LIN {X 0,Y 608.989,Z 328.359,A -85,B 0,C 180,E1 28957.914,E2 28957.914} C_VEL
LIN {X 0,Y 609.026,Z 328.336,A -85,B 0,C 180,E1 28955.043,E2 28955.043} C_VEL
LIN {X 0,Y 608.99,Z 328.372,A -85,B 0,C 180,E1 28951.886,E2 28951.886} C_VEL
LIN {X 0,Y 608.992,Z 328.336,A -85,B 0,C 180,E1 28949.168,E2 28949.168} C_VEL
LIN {X 0,Y 608.991,Z 328.34,A -85,B 0,C 180,E1 28945.952,E2 28945.952} C_VEL
LIN {X 0,Y 609.049,Z 328.447,A -85,B 0,C 180,E1 28944.672,E2 28944.672} C_VEL
LIN {X 0,Y 610.191,Z 331.571,A -85,B 0,C 180,E1 28944.457,E2 28944.457} C_VEL
LIN {X 0,Y 612.692,Z 334.142,A -85,B 0,C 180,E1 28944.077,E2 28944.077} C_VEL
LIN {X 0,Y 613.552,Z 335.036,A -85,B 0,C 180,E1 28943.948,E2 28943.948} C_VEL
LIN {X 0,Y 616.041,Z 338.824,A -85,B 0,C 180,E1 28943.555,E2 28943.555} C_VEL
LIN {X 0,Y 618.268,Z 341.03,A -85,B 0,C 180,E1 28943.231,E2 28943.231} C_VEL
LIN {X 0,Y 621.516,Z 345.277,A -85,B 0,C 180,E1 28942.749,E2 28942.749} C_VEL
LIN {X 0,Y 626.243,Z 351.226,A -85,B 0,C 180,E1 28942.069,E2 28942.069} C_VEL
LIN {X 0,Y 641.999,Z 372.195,A -85,B 0,C 180,E1 28939.923,E2 28939.923} C_VEL
LIN {X 0,Y 650.667,Z 384.496,A -85,B 0,C 180,E1 28938.812,E2 28938.812} C_VEL
LIN {X 0,Y 648.081,Z 493.94,A -85,B 0,C 180,E1 28937.285,E2 28937.285} C_VEL
LIN {X 0,Y 647.227,Z 501.644,A -85,B 0,C 180,E1 28937.244,E2 28937.244} C_VEL
LIN {X 0,Y 642.505,Z 522.314,A -85,B 0,C 180,E1 28937.368,E2 28937.368} C_VEL
LIN {X 0,Y 641.836,Z 528.923,A -85,B 0,C 180,E1 28937.326,E2 28937.326} C_VEL
LIN {X 0,Y 636.639,Z 753.083,A -85,B 0,C 180,E1 28934.254,E2 28934.254} C_VEL
LIN {X 0,Y 635.306,Z 802.32,A -85,B 0,C 180,E1 28933.564,E2 28933.564} C_VEL
LIN {X 0,Y 633.786,Z 830.264,A -85,B 0,C 180,E1 28933.009,E2 28933.009} C_VEL
LIN {X 0,Y 632.226,Z 852.784,A -85,B 0,C 180,E1 28932.423,E2 28932.423} C_VEL
LIN {X 0,Y 630.535,Z 873.77,A -85,B 0,C 180,E1 28931.759,E2 28931.759} C_VEL
LIN {X 0,Y 628.677,Z 894.198,A -85,B 0,C 180,E1 28930.999,E2 28930.999} C_VEL
LIN {X 0,Y 626.241,Z 918.774,A -85,B 0,C 180,E1 28929.929,E2 28929.929} C_VEL
LIN {X 0,Y 623.465,Z 943.532,A -85,B 0,C 180,E1 28928.644,E2 28928.644} C_VEL
LIN {X 0,Y 621.108,Z 963.324,A -85,B 0,C 180,E1 28927.471,E2 28927.471} C_VEL
LIN {X 0,Y 618.751,Z 982.414,A -85,B 0,C 180,E1 28926.201,E2 28926.201} C_VEL
LIN {X 0,Y 616.012,Z 1004.354,A -85,B 0,C 180,E1 28924.561,E2 28924.561} C_VEL
LIN {X 0,Y 613.186,Z 1025.937,A -85,B 0,C 180,E1 28922.71,E2 28922.71} C_VEL
LIN {X 0,Y 611.026,Z 1042.889,A -85,B 0,C 180,E1 28921.082,E2 28921.082} C_VEL
LIN {X 0,Y 608.96,Z 1059.696,A -85,B 0,C 180,E1 28919.294,E2 28919.294} C_VEL
LIN {X 0,Y 606.611,Z 1079.55,A -85,B 0,C 180,E1 28916.906,E2 28916.906} C_VEL
LIN {X 0,Y 604.981,Z 1094.558,A -85,B 0,C 180,E1 28914.855,E2 28914.855} C_VEL
LIN {X 0,Y 603.522,Z 1109.273,A -85,B 0,C 180,E1 28912.604,E2 28912.604} C_VEL
LIN {X 0,Y 602.265,Z 1123.493,A -85,B 0,C 180,E1 28910.1,E2 28910.1} C_VEL
LIN {X 0,Y 601.47,Z 1133.871,A -85,B 0,C 180,E1 28908.011,E2 28908.011} C_VEL
LIN {X 0,Y 600.869,Z 1143.337,A -85,B 0,C 180,E1 28905.837,E2 28905.837} C_VEL
LIN {X 0,Y 600.412,Z 1152.859,A -85,B 0,C 180,E1 28903.286,E2 28903.286} C_VEL
LIN {X 0,Y 600.121,Z 1160.474,A -85,B 0,C 180,E1 28900.755,E2 28900.755} C_VEL
LIN {X 0,Y 600.004,Z 1166.042,A -85,B 0,C 180,E1 28898.433,E2 28898.433} C_VEL
LIN {X 0,Y 599.936,Z 1170.564,A -85,B 0,C 180,E1 28895.931,E2 28895.931} C_VEL
LIN {X 0,Y 599.914,Z 1173.552,A -85,B 0,C 180,E1 28893.344,E2 28893.344} C_VEL
LIN {X 0,Y 599.91,Z 1174.749,A -85,B 0,C 180,E1 28891.05,E2 28891.05} C_VEL
LIN {X 0,Y 599.907,Z 1174.793,A -85,B 0,C 180,E1 28889.045,E2 28889.045} C_VEL
LIN {X 0,Y 599.913,Z 1173.823,A -85,B 0,C 180,E1 28886.943,E2 28886.943} C_VEL
LIN {X 0,Y 599.923,Z 1171.362,A -85,B 0,C 180,E1 28884.549,E2 28884.549} C_VEL
LIN {X 0,Y 599.991,Z 1166.847,A -85,B 0,C 180,E1 28881.855,E2 28881.855} C_VEL
LIN {X 0,Y 600.108,Z 1161.212,A -85,B 0,C 180,E1 28879.437,E2 28879.437} C_VEL
LIN {X 0,Y 600.366,Z 1154.109,A -85,B 0,C 180,E1 28877.007,E2 28877.007} C_VEL
LIN {X 0,Y 600.82,Z 1144.11,A -85,B 0,C 180,E1 28874.261,E2 28874.261} C_VEL
LIN {X 0,Y 601.415,Z 1134.739,A -85,B 0,C 180,E1 28872.088,E2 28872.088} C_VEL
LIN {X 0,Y 602.187,Z 1124.472,A -85,B 0,C 180,E1 28869.999,E2 28869.999} C_VEL
LIN {X 0,Y 603.358,Z 1111.046,A -85,B 0,C 180,E1 28867.595,E2 28867.595} C_VEL
LIN {X 0,Y 604.905,Z 1095.289,A -85,B 0,C 180,E1 28865.16,E2 28865.16} C_VEL
LIN {X 0,Y 606.386,Z 1081.406,A -85,B 0,C 180,E1 28863.247,E2 28863.247} C_VEL
LIN {X 0,Y 608.474,Z 1064.093,A -85,B 0,C 180,E1 28861.112,E2 28861.112} C_VEL
LIN {X 0,Y 610.807,Z 1044.692,A -85,B 0,C 180,E1 28859.01,E2 28859.01} C_VEL
LIN {X 0,Y 612.933,Z 1027.84,A -85,B 0,C 180,E1 28857.375,E2 28857.375} C_VEL
LIN {X 0,Y 615.269,Z 1009.673,A -85,B 0,C 180,E1 28855.787,E2 28855.787} C_VEL
LIN {X 0,Y 618.361,Z 985.78,A -85,B 0,C 180,E1 28853.945,E2 28853.945} C_VEL
LIN {X 0,Y 620.892,Z 965.162,A -85,B 0,C 180,E1 28852.555,E2 28852.555} C_VEL
LIN {X 0,Y 623.12,Z 946.531,A -85,B 0,C 180,E1 28851.436,E2 28851.436} C_VEL
LIN {X 0,Y 625.266,Z 927.631,A -85,B 0,C 180,E1 28850.425,E2 28850.425} C_VEL
LIN {X 0,Y 627.464,Z 906.92,A -85,B 0,C 180,E1 28849.448,E2 28849.448} C_VEL
LIN {X 0,Y 629.999,Z 880.352,A -85,B 0,C 180,E1 28848.378,E2 28848.378} C_VEL
LIN {X 0,Y 631.987,Z 855.974,A -85,B 0,C 180,E1 28847.58,E2 28847.58} C_VEL
LIN {X 0,Y 633.509,Z 834.338,A -85,B 0,C 180,E1 28846.999,E2 28846.999} C_VEL
LIN {X 0,Y 634.765,Z 812.654,A -85,B 0,C 180,E1 28846.532,E2 28846.532} C_VEL
LIN {X 0,Y 635.903,Z 785.947,A -85,B 0,C 180,E1 28846.1,E2 28846.1} C_VEL
LIN {X 0,Y 641.062,Z 561.333,A -85,B 0,C 180,E1 28843.033,E2 28843.033} C_VEL
LIN {X 0,Y 645.263,Z 388.229,A -85,B 0,C 180,E1 28840.604,E2 28840.604} C_VEL
LIN {X 0,Y 633.126,Z 371.566,A -85,B 0,C 180,E1 28839.002,E2 28839.002} C_VEL
LIN {X 0,Y 622.468,Z 357.45,A -85,B 0,C 180,E1 28837.503,E2 28837.503} C_VEL
LIN {X 0,Y 617.121,Z 350.737,A -85,B 0,C 180,E1 28836.718,E2 28836.718} C_VEL
LIN {X 0,Y 613.975,Z 346.647,A -85,B 0,C 180,E1 28836.24,E2 28836.24} C_VEL
LIN {X 0,Y 610.658,Z 342.52,A -85,B 0,C 180,E1 28835.728,E2 28835.728} C_VEL
LIN {X 0,Y 609.495,Z 340.975,A -85,B 0,C 180,E1 28835.544,E2 28835.544} C_VEL
LIN {X 0,Y 606.547,Z 337.524,A -85,B 0,C 180,E1 28835.079,E2 28835.079} C_VEL
LIN {X 0,Y 605.262,Z 335.42,A -85,B 0,C 180,E1 28834.861,E2 28834.861} C_VEL
LIN {X 0,Y 602.43,Z 332.951,A -85,B 0,C 180,E1 28834.419,E2 28834.419} C_VEL
LIN {X 0,Y 601.129,Z 329.909,A -85,B 0,C 180,E1 28834.172,E2 28834.172} C_VEL
LIN {X 0,Y 601.037,Z 329.326,A -85,B 0,C 180,E1 28834.133,E2 28834.133} C_VEL
LIN {X 0,Y 601.047,Z 329.325,A -85,B 0,C 180,E1 28830.823,E2 28830.823} C_VEL
LIN {X 0,Y 601.042,Z 329.362,A -85,B 0,C 180,E1 28828.086,E2 28828.086} C_VEL
LIN {X 0,Y 601.077,Z 329.323,A -85,B 0,C 180,E1 28824.889,E2 28824.889} C_VEL
LIN {X 0,Y 601.044,Z 329.352,A -85,B 0,C 180,E1 28822.084,E2 28822.084} C_VEL
LIN {X 0,Y 601.118,Z 329.326,A -85,B 0,C 180,E1 28819.028,E2 28819.028} C_VEL
LIN {X 0,Y 601.048,Z 329.337,A -85,B 0,C 180,E1 28816.031,E2 28816.031} C_VEL
LIN {X 0,Y 601.129,Z 329.335,A -85,B 0,C 180,E1 28812.977,E2 28812.977} C_VEL
LIN {X 0,Y 601.054,Z 329.33,A -85,B 0,C 180,E1 28809.963,E2 28809.963} C_VEL
LIN {X 0,Y 601.14,Z 329.337,A -85,B 0,C 180,E1 28806.878,E2 28806.878} C_VEL
LIN {X 0,Y 601.059,Z 329.328,A -85,B 0,C 180,E1 28803.815,E2 28803.815} C_VEL
LIN {X 0,Y 601.136,Z 329.337,A -85,B 0,C 180,E1 28800.762,E2 28800.762} C_VEL
LIN {X 0,Y 601.067,Z 329.327,A -85,B 0,C 180,E1 28797.712,E2 28797.712} C_VEL
LIN {X 0,Y 601.134,Z 329.338,A -85,B 0,C 180,E1 28794.655,E2 28794.655} C_VEL
LIN {X 0,Y 601.073,Z 329.323,A -85,B 0,C 180,E1 28791.582,E2 28791.582} C_VEL
LIN {X 0,Y 601.137,Z 329.345,A -85,B 0,C 180,E1 28788.486,E2 28788.486} C_VEL
LIN {X 0,Y 601.077,Z 329.316,A -85,B 0,C 180,E1 28785.354,E2 28785.354} C_VEL
LIN {X 0,Y 601.14,Z 329.351,A -85,B 0,C 180,E1 28782.279,E2 28782.279} C_VEL
LIN {X 0,Y 601.085,Z 329.318,A -85,B 0,C 180,E1 28779.146,E2 28779.146} C_VEL
LIN {X 0,Y 601.136,Z 329.331,A -85,B 0,C 180,E1 28776.055,E2 28776.055} C_VEL
LIN {X 0,Y 601.096,Z 329.352,A -85,B 0,C 180,E1 28772.884,E2 28772.884} C_VEL
LIN {X 0,Y 601.136,Z 329.316,A -85,B 0,C 180,E1 28769.682,E2 28769.682} C_VEL
LIN {X 0,Y 601.155,Z 329.494,A -85,B 0,C 180,E1 28767.73,E2 28767.73} C_VEL
LIN {X 0,Y 602.27,Z 332.603,A -85,B 0,C 180,E1 28767.233,E2 28767.233} C_VEL
LIN {X 0,Y 603.588,Z 334.345,A -85,B 0,C 180,E1 28766.861,E2 28766.861} C_VEL
LIN {X 0,Y 605.493,Z 338.277,A -85,B 0,C 180,E1 28766.185,E2 28766.185} C_VEL
LIN {X 0,Y 610.426,Z 347.698,A -85,B 0,C 180,E1 28764.617,E2 28764.617} C_VEL
LIN {X 0,Y 625.354,Z 368.362,A -85,B 0,C 180,E1 28762.368,E2 28762.368} C_VEL
LIN {X 0,Y 641.991,Z 392.611,A -85,B 0,C 180,E1 28760.082,E2 28760.082} C_VEL
LIN {X 0,Y 645.613,Z 398.452,A -85,B 0,C 180,E1 28759.605,E2 28759.605} C_VEL
LIN {X 0,Y 640.632,Z 604.673,A -85,B 0,C 180,E1 28756.729,E2 28756.729} C_VEL
LIN {X 0,Y 635.662,Z 822.347,A -85,B 0,C 180,E1 28753.759,E2 28753.759} C_VEL
LIN {X 0,Y 634.658,Z 844.67,A -85,B 0,C 180,E1 28753.384,E2 28753.384} C_VEL
LIN {X 0,Y 633.39,Z 866.16,A -85,B 0,C 180,E1 28752.912,E2 28752.912} C_VEL
LIN {X 0,Y 631.712,Z 889.713,A -85,B 0,C 180,E1 28752.266,E2 28752.266} C_VEL
LIN {X 0,Y 629.333,Z 917.45,A -85,B 0,C 180,E1 28751.31,E2 28751.31} C_VEL
LIN {X 0,Y 627.184,Z 939.464,A -85,B 0,C 180,E1 28750.394,E2 28750.394} C_VEL
LIN {X 0,Y 625.147,Z 958.693,A -85,B 0,C 180,E1 28749.476,E2 28749.476} C_VEL
LIN {X 0,Y 622.955,Z 977.953,A -85,B 0,C 180,E1 28748.438,E2 28748.438} C_VEL
LIN {X 0,Y 620.583,Z 997.794,A -85,B 0,C 180,E1 28747.234,E2 28747.234} C_VEL
LIN {X 0,Y 617.516,Z 1022.228,A -85,B 0,C 180,E1 28745.54,E2 28745.54} C_VEL
LIN {X 0,Y 614.967,Z 1041.908,A -85,B 0,C 180,E1 28743.981,E2 28743.981} C_VEL
LIN {X 0,Y 612.783,Z 1059.055,A -85,B 0,C 180,E1 28742.467,E2 28742.467} C_VEL
LIN {X 0,Y 610.531,Z 1077.071,A -85,B 0,C 180,E1 28740.704,E2 28740.704} C_VEL
LIN {X 0,Y 608.06,Z 1097.15,A -85,B 0,C 180,E1 28738.48,E2 28738.48} C_VEL
LIN {X 0,Y 606.258,Z 1112.619,A -85,B 0,C 180,E1 28736.547,E2 28736.547} C_VEL
LIN {X 0,Y 604.639,Z 1127.891,A -85,B 0,C 180,E1 28734.419,E2 28734.419} C_VEL
LIN {X 0,Y 603.102,Z 1143.702,A -85,B 0,C 180,E1 28731.902,E2 28731.902} C_VEL
LIN {X 0,Y 602.121,Z 1155.273,A -85,B 0,C 180,E1 28729.801,E2 28729.801} C_VEL
LIN {X 0,Y 601.343,Z 1165.909,A -85,B 0,C 180,E1 28727.615,E2 28727.615} C_VEL
LIN {X 0,Y 600.69,Z 1177.02,A -85,B 0,C 180,E1 28724.951,E2 28724.951} C_VEL
LIN {X 0,Y 600.299,Z 1185.324,A -85,B 0,C 180,E1 28722.557,E2 28722.557} C_VEL
LIN {X 0,Y 600.092,Z 1191.863,A -85,B 0,C 180,E1 28720.27,E2 28720.27} C_VEL
LIN {X 0,Y 599.973,Z 1197.542,A -85,B 0,C 180,E1 28717.758,E2 28717.758} C_VEL
LIN {X 0,Y 599.926,Z 1201.663,A -85,B 0,C 180,E1 28715.163,E2 28715.163} C_VEL
LIN {X 0,Y 599.915,Z 1203.927,A -85,B 0,C 180,E1 28712.866,E2 28712.866} C_VEL
LIN {X 0,Y 599.895,Z 1204.849,A -85,B 0,C 180,E1 28710.668,E2 28710.668} C_VEL
LIN {X 0,Y 599.908,Z 1204.623,A -85,B 0,C 180,E1 28708.376,E2 28708.376} C_VEL
LIN {X 0,Y 599.918,Z 1202.789,A -85,B 0,C 180,E1 28705.795,E2 28705.795} C_VEL
LIN {X 0,Y 599.944,Z 1199.513,A -85,B 0,C 180,E1 28703.375,E2 28703.375} C_VEL
LIN {X 0,Y 600.014,Z 1195.106,A -85,B 0,C 180,E1 28701.085,E2 28701.085} C_VEL
LIN {X 0,Y 600.197,Z 1188.477,A -85,B 0,C 180,E1 28698.469,E2 28698.469} C_VEL
LIN {X 0,Y 600.504,Z 1180.572,A -85,B 0,C 180,E1 28696.029,E2 28696.029} C_VEL
LIN {X 0,Y 600.938,Z 1172.306,A -85,B 0,C 180,E1 28693.868,E2 28693.868} C_VEL
LIN {X 0,Y 601.566,Z 1162.692,A -85,B 0,C 180,E1 28691.691,E2 28691.691} C_VEL
LIN {X 0,Y 602.621,Z 1149.398,A -85,B 0,C 180,E1 28689.092,E2 28689.092} C_VEL
LIN {X 0,Y 603.843,Z 1135.741,A -85,B 0,C 180,E1 28686.791,E2 28686.791} C_VEL
LIN {X 0,Y 605.279,Z 1121.578,A -85,B 0,C 180,E1 28684.669,E2 28684.669} C_VEL
LIN {X 0,Y 607.376,Z 1103.066,A -85,B 0,C 180,E1 28682.233,E2 28682.233} C_VEL
LIN {X 0,Y 609.273,Z 1086.965,A -85,B 0,C 180,E1 28680.359,E2 28680.359} C_VEL
LIN {X 0,Y 611.356,Z 1070.397,A -85,B 0,C 180,E1 28678.622,E2 28678.622} C_VEL
LIN {X 0,Y 614.09,Z 1049.297,A -85,B 0,C 180,E1 28676.647,E2 28676.647} C_VEL
LIN {X 0,Y 616.657,Z 1028.87,A -85,B 0,C 180,E1 28674.969,E2 28674.969} C_VEL
LIN {X 0,Y 619.038,Z 1009.978,A -85,B 0,C 180,E1 28673.583,E2 28673.583} C_VEL
LIN {X 0,Y 621.631,Z 988.944,A -85,B 0,C 180,E1 28672.207,E2 28672.207} C_VEL
LIN {X 0,Y 624.587,Z 963.722,A -85,B 0,C 180,E1 28670.778,E2 28670.778} C_VEL
LIN {X 0,Y 626.818,Z 942.858,A -85,B 0,C 180,E1 28669.757,E2 28669.757} C_VEL
LIN {X 0,Y 628.829,Z 922.588,A -85,B 0,C 180,E1 28668.892,E2 28668.892} C_VEL
LIN {X 0,Y 630.688,Z 901.904,A -85,B 0,C 180,E1 28668.131,E2 28668.131} C_VEL
LIN {X 0,Y 632.495,Z 879.261,A -85,B 0,C 180,E1 28667.429,E2 28667.429} C_VEL
LIN {X 0,Y 634.363,Z 850.617,A -85,B 0,C 180,E1 28666.733,E2 28666.733} C_VEL
LIN {X 0,Y 635.496,Z 826.763,A -85,B 0,C 180,E1 28666.307,E2 28666.307} C_VEL
LIN {X 0,Y 639.752,Z 643.039,A -85,B 0,C 180,E1 28663.798,E2 28663.798} C_VEL
LIN {X 0,Y 644.902,Z 427.367,A -85,B 0,C 180,E1 28660.804,E2 28660.804} C_VEL
LIN {X 0,Y 645.53,Z 398.043,A -85,B 0,C 180,E1 28660.38,E2 28660.38} C_VEL
LIN {X 0,Y 628.947,Z 373.409,A -85,B 0,C 180,E1 28658.144,E2 28658.144} C_VEL
LIN {X 0,Y 616.881,Z 356.682,A -85,B 0,C 180,E1 28656.388,E2 28656.388} C_VEL
LIN {X 0,Y 609.775,Z 346.816,A -85,B 0,C 180,E1 28655.254,E2 28655.254} C_VEL
LIN {X 0,Y 605.475,Z 338.255,A -85,B 0,C 180,E1 28653.816,E2 28653.816} C_VEL
LIN {X 0,Y 603.577,Z 334.304,A -85,B 0,C 180,E1 28653.14,E2 28653.14} C_VEL
LIN {X 0,Y 601.478,Z 330.889,A -85,B 0,C 180,E1 28652.477,E2 28652.477} C_VEL
LIN {X 0,Y 601.135,Z 329.344,A -85,B 0,C 180,E1 28652.215,E2 28652.215} C_VEL
LIN {X 0,Y 601.094,Z 329.323,A -85,B 0,C 180,E1 28649.06,E2 28649.06} C_VEL
LIN {X 0,Y 601.134,Z 329.317,A -85,B 0,C 180,E1 28645.942,E2 28645.942} C_VEL
LIN {X 0,Y 601.093,Z 329.356,A -85,B 0,C 180,E1 28642.804,E2 28642.804} C_VEL
LIN {X 0,Y 601.133,Z 329.312,A -85,B 0,C 180,E1 28639.633,E2 28639.633} C_VEL
LIN {X 0,Y 601.089,Z 329.346,A -85,B 0,C 180,E1 28636.526,E2 28636.526} C_VEL
LIN {X 0,Y 601.127,Z 329.33,A -85,B 0,C 180,E1 28633.337,E2 28633.337} C_VEL
LIN {X 0,Y 601.082,Z 329.332,A -85,B 0,C 180,E1 28630.35,E2 28630.35} C_VEL
LIN {X 0,Y 601.122,Z 329.339,A -85,B 0,C 180,E1 28627.167,E2 28627.167} C_VEL
LIN {X 0,Y 601.077,Z 329.327,A -85,B 0,C 180,E1 28624.197,E2 28624.197} C_VEL
LIN {X 0,Y 601.109,Z 329.345,A -85,B 0,C 180,E1 28620.953,E2 28620.953} C_VEL
LIN {X 0,Y 601.07,Z 329.328,A -85,B 0,C 180,E1 28618.093,E2 28618.093} C_VEL
LIN {X 0,Y 601.117,Z 329.342,A -85,B 0,C 180,E1 28614.942,E2 28614.942} C_VEL
LIN {X 0,Y 601.061,Z 329.33,A -85,B 0,C 180,E1 28612.064,E2 28612.064} C_VEL
LIN {X 0,Y 601.124,Z 329.341,A -85,B 0,C 180,E1 28608.918,E2 28608.918} C_VEL
LIN {X 0,Y 601.056,Z 329.325,A -85,B 0,C 180,E1 28605.888,E2 28605.888} C_VEL
LIN {X 0,Y 601.122,Z 329.349,A -85,B 0,C 180,E1 28602.778,E2 28602.778} C_VEL
LIN {X 0,Y 601.049,Z 329.318,A -85,B 0,C 180,E1 28599.755,E2 28599.755} C_VEL
LIN {X 0,Y 601.122,Z 329.353,A -85,B 0,C 180,E1 28596.657,E2 28596.657} C_VEL
LIN {X 0,Y 601.044,Z 329.328,A -85,B 0,C 180,E1 28593.629,E2 28593.629} C_VEL
LIN {X 0,Y 601.127,Z 329.322,A -85,B 0,C 180,E1 28590.614,E2 28590.614} C_VEL
LIN {X 0,Y 601.039,Z 329.365,A -85,B 0,C 180,E1 28587.61,E2 28587.61} C_VEL
LIN {X 0,Y 601.062,Z 329.488,A -85,B 0,C 180,E1 28585.75,E2 28585.75} C_VEL
LIN {X 0,Y 602.122,Z 332.471,A -85,B 0,C 180,E1 28585.538,E2 28585.538} C_VEL
LIN {X 0,Y 604.551,Z 334.996,A -85,B 0,C 180,E1 28585.149,E2 28585.149} C_VEL
LIN {X 0,Y 605.796,Z 336.054,A -85,B 0,C 180,E1 28584.957,E2 28584.957} C_VEL
LIN {X 0,Y 608.346,Z 339.929,A -85,B 0,C 180,E1 28584.535,E2 28584.535} C_VEL
LIN {X 0,Y 610.44,Z 342.145,A -85,B 0,C 180,E1 28584.214,E2 28584.214} C_VEL
LIN {X 0,Y 613.674,Z 346.372,A -85,B 0,C 180,E1 28583.711,E2 28583.711} C_VEL
LIN {X 0,Y 615.392,Z 348.396,A -85,B 0,C 180,E1 28583.452,E2 28583.452} C_VEL
LIN {X 0,Y 620.152,Z 354.623,A -85,B 0,C 180,E1 28582.74,E2 28582.74} C_VEL
LIN {X 0,Y 627.738,Z 364.357,A -85,B 0,C 180,E1 28581.653,E2 28581.653} C_VEL
LIN {X 0,Y 638.992,Z 379.544,A -85,B 0,C 180,E1 28580.12,E2 28580.12} C_VEL
LIN {X 0,Y 645.334,Z 388.642,A -85,B 0,C 180,E1 28579.292,E2 28579.292} C_VEL
LIN {X 0,Y 641.836,Z 528.923,A -85,B 0,C 180,E1 28577.326,E2 28577.326} C_VEL
LIN {X 0,Y 640.974,Z 536.628,A -85,B 0,C 180,E1 28577.285,E2 28577.285} C_VEL
LIN {X 0,Y 636.236,Z 557.294,A -85,B 0,C 180,E1 28577.413,E2 28577.413} C_VEL
LIN {X 0,Y 635.561,Z 563.903,A -85,B 0,C 180,E1 28577.372,E2 28577.372} C_VEL
LIN {X 0,Y 630.023,Z 789.388,A -85,B 0,C 180,E1 28574.266,E2 28574.266} C_VEL
LIN {X 0,Y 628.918,Z 813.43,A -85,B 0,C 180,E1 28573.868,E2 28573.868} C_VEL
LIN {X 0,Y 627.63,Z 834.391,A -85,B 0,C 180,E1 28573.413,E2 28573.413} C_VEL
LIN {X 0,Y 626.015,Z 856.115,A -85,B 0,C 180,E1 28572.825,E2 28572.825} C_VEL
LIN {X 0,Y 623.994,Z 879.701,A -85,B 0,C 180,E1 28572.05,E2 28572.05} C_VEL
LIN {X 0,Y 621.328,Z 906.369,A -85,B 0,C 180,E1 28570.977,E2 28570.977} C_VEL
LIN {X 0,Y 619.027,Z 926.941,A -85,B 0,C 180,E1 28570.005,E2 28570.005} C_VEL
LIN {X 0,Y 616.731,Z 946.061,A -85,B 0,C 180,E1 28568.979,E2 28568.979} C_VEL
LIN {X 0,Y 614.362,Z 964.812,A -85,B 0,C 180,E1 28567.847,E2 28567.847} C_VEL
LIN {X 0,Y 611.778,Z 984.623,A -85,B 0,C 180,E1 28566.506,E2 28566.506} C_VEL
LIN {X 0,Y 608.522,Z 1008.702,A -85,B 0,C 180,E1 28564.646,E2 28564.646} C_VEL
LIN {X 0,Y 605.936,Z 1027.5,A -85,B 0,C 180,E1 28562.993,E2 28562.993} C_VEL
LIN {X 0,Y 603.65,Z 1044.414,A -85,B 0,C 180,E1 28561.338,E2 28561.338} C_VEL
LIN {X 0,Y 601.218,Z 1063.385,A -85,B 0,C 180,E1 28559.271,E2 28559.271} C_VEL
LIN {X 0,Y 598.985,Z 1080.753,A -85,B 0,C 180,E1 28557.11,E2 28557.11} C_VEL
LIN {X 0,Y 597.346,Z 1094.79,A -85,B 0,C 180,E1 28555.16,E2 28555.16} C_VEL
LIN {X 0,Y 595.793,Z 1109.519,A -85,B 0,C 180,E1 28552.874,E2 28552.874} C_VEL
LIN {X 0,Y 594.458,Z 1123.498,A -85,B 0,C 180,E1 28550.375,E2 28550.375} C_VEL
LIN {X 0,Y 593.579,Z 1134.218,A -85,B 0,C 180,E1 28548.182,E2 28548.182} C_VEL
LIN {X 0,Y 592.951,Z 1143.498,A -85,B 0,C 180,E1 28546.014,E2 28546.014} C_VEL
LIN {X 0,Y 592.439,Z 1153.181,A -85,B 0,C 180,E1 28543.369,E2 28543.369} C_VEL
LIN {X 0,Y 592.131,Z 1160.727,A -85,B 0,C 180,E1 28540.803,E2 28540.803} C_VEL
LIN {X 0,Y 592.008,Z 1166.247,A -85,B 0,C 180,E1 28538.449,E2 28538.449} C_VEL
LIN {X 0,Y 591.937,Z 1170.713,A -85,B 0,C 180,E1 28535.914,E2 28535.914} C_VEL
LIN {X 0,Y 591.915,Z 1173.621,A -85,B 0,C 180,E1 28533.291,E2 28533.291} C_VEL
LIN {X 0,Y 591.91,Z 1174.749,A -85,B 0,C 180,E1 28531.065,E2 28531.065} C_VEL
LIN {X 0,Y 591.907,Z 1174.792,A -85,B 0,C 180,E1 28529.032,E2 28529.032} C_VEL
LIN {X 0,Y 591.913,Z 1173.82,A -85,B 0,C 180,E1 28526.901,E2 28526.901} C_VEL
LIN {X 0,Y 591.925,Z 1171.361,A -85,B 0,C 180,E1 28524.475,E2 28524.475} C_VEL
LIN {X 0,Y 591.996,Z 1166.85,A -85,B 0,C 180,E1 28521.746,E2 28521.746} C_VEL
LIN {X 0,Y 592.118,Z 1161.383,A -85,B 0,C 180,E1 28519.361,E2 28519.361} C_VEL
LIN {X 0,Y 592.377,Z 1154.711,A -85,B 0,C 180,E1 28517.027,E2 28517.027} C_VEL
LIN {X 0,Y 592.856,Z 1144.917,A -85,B 0,C 180,E1 28514.245,E2 28514.245} C_VEL
LIN {X 0,Y 593.509,Z 1135.193,A -85,B 0,C 180,E1 28511.942,E2 28511.942} C_VEL
LIN {X 0,Y 594.33,Z 1124.982,A -85,B 0,C 180,E1 28509.826,E2 28509.826} C_VEL
LIN {X 0,Y 595.458,Z 1112.791,A -85,B 0,C 180,E1 28507.594,E2 28507.594} C_VEL
LIN {X 0,Y 597.141,Z 1096.786,A -85,B 0,C 180,E1 28505.042,E2 28505.042} C_VEL
LIN {X 0,Y 598.708,Z 1082.94,A -85,B 0,C 180,E1 28503.091,E2 28503.091} C_VEL
LIN {X 0,Y 600.532,Z 1068.342,A -85,B 0,C 180,E1 28501.238,E2 28501.238} C_VEL
LIN {X 0,Y 603.061,Z 1049.29,A -85,B 0,C 180,E1 28499.071,E2 28499.071} C_VEL
LIN {X 0,Y 605.661,Z 1029.497,A -85,B 0,C 180,E1 28497.103,E2 28497.103} C_VEL
LIN {X 0,Y 608.025,Z 1012.098,A -85,B 0,C 180,E1 28495.55,E2 28495.55} C_VEL
LIN {X 0,Y 610.886,Z 991.408,A -85,B 0,C 180,E1 28493.898,E2 28493.898} C_VEL
LIN {X 0,Y 614.013,Z 967.68,A -85,B 0,C 180,E1 28492.246,E2 28492.246} C_VEL
LIN {X 0,Y 616.463,Z 948.317,A -85,B 0,C 180,E1 28491.061,E2 28491.061} C_VEL
LIN {X 0,Y 618.746,Z 929.337,A -85,B 0,C 180,E1 28490.028,E2 28490.028} C_VEL
LIN {X 0,Y 620.882,Z 910.294,A -85,B 0,C 180,E1 28489.109,E2 28489.109} C_VEL
LIN {X 0,Y 623.003,Z 889.668,A -85,B 0,C 180,E1 28488.239,E2 28488.239} C_VEL
LIN {X 0,Y 625.236,Z 865.972,A -85,B 0,C 180,E1 28487.388,E2 28487.388} C_VEL
LIN {X 0,Y 627.373,Z 838.238,A -85,B 0,C 180,E1 28486.592,E2 28486.592} C_VEL
LIN {X 0,Y 628.761,Z 816.335,A -85,B 0,C 180,E1 28486.099,E2 28486.099} C_VEL
LIN {X 0,Y 629.814,Z 794.671,A -85,B 0,C 180,E1 28485.724,E2 28485.724} C_VEL
LIN {X 0,Y 635.163,Z 579.694,A -85,B 0,C 180,E1 28482.758,E2 28482.758} C_VEL
LIN {X 0,Y 639.979,Z 392.395,A -85,B 0,C 180,E1 28480.117,E2 28480.117} C_VEL
LIN {X 0,Y 628.585,Z 376.663,A -85,B 0,C 180,E1 28478.576,E2 28478.576} C_VEL
LIN {X 0,Y 618.701,Z 363.583,A -85,B 0,C 180,E1 28477.159,E2 28477.159} C_VEL
LIN {X 0,Y 610.545,Z 353.158,A -85,B 0,C 180,E1 28475.924,E2 28475.924} C_VEL
LIN {X 0,Y 606.961,Z 348.407,A -85,B 0,C 180,E1 28475.355,E2 28475.355} C_VEL
LIN {X 0,Y 603.197,Z 343.928,A -85,B 0,C 180,E1 28474.752,E2 28474.752} C_VEL
LIN {X 0,Y 602.018,Z 342.306,A -85,B 0,C 180,E1 28474.555,E2 28474.555} C_VEL
LIN {X 0,Y 598.977,Z 339.128,A -85,B 0,C 180,E1 28474.06,E2 28474.06} C_VEL
LIN {X 0,Y 597.576,Z 336.526,A -85,B 0,C 180,E1 28473.804,E2 28473.804} C_VEL
LIN {X 0,Y 594.664,Z 334.086,A -85,B 0,C 180,E1 28473.327,E2 28473.327} C_VEL
LIN {X 0,Y 593.275,Z 331.155,A -85,B 0,C 180,E1 28473.056,E2 28473.056} C_VEL
LIN {X 0,Y 593.122,Z 330.336,A -85,B 0,C 180,E1 28472.992,E2 28472.992} C_VEL
LIN {X 0,Y 593.094,Z 330.31,A -85,B 0,C 180,E1 28470.137,E2 28470.137} C_VEL
LIN {X 0,Y 593.14,Z 330.328,A -85,B 0,C 180,E1 28466.967,E2 28466.967} C_VEL
LIN {X 0,Y 593.103,Z 330.333,A -85,B 0,C 180,E1 28464.078,E2 28464.078} C_VEL
LIN {X 0,Y 593.163,Z 330.301,A -85,B 0,C 180,E1 28460.958,E2 28460.958} C_VEL
LIN {X 0,Y 593.111,Z 330.348,A -85,B 0,C 180,E1 28457.969,E2 28457.969} C_VEL
LIN {X 0,Y 593.173,Z 330.297,A -85,B 0,C 180,E1 28454.846,E2 28454.846} C_VEL
LIN {X 0,Y 593.117,Z 330.348,A -85,B 0,C 180,E1 28451.869,E2 28451.869} C_VEL
LIN {X 0,Y 593.181,Z 330.295,A -85,B 0,C 180,E1 28448.726,E2 28448.726} C_VEL
LIN {X 0,Y 593.123,Z 330.347,A -85,B 0,C 180,E1 28445.805,E2 28445.805} C_VEL
LIN {X 0,Y 593.189,Z 330.293,A -85,B 0,C 180,E1 28442.705,E2 28442.705} C_VEL
LIN {X 0,Y 593.129,Z 330.346,A -85,B 0,C 180,E1 28439.614,E2 28439.614} C_VEL
LIN {X 0,Y 593.19,Z 330.293,A -85,B 0,C 180,E1 28436.521,E2 28436.521} C_VEL
LIN {X 0,Y 593.137,Z 330.345,A -85,B 0,C 180,E1 28433.418,E2 28433.418} C_VEL
LIN {X 0,Y 593.19,Z 330.296,A -85,B 0,C 180,E1 28430.296,E2 28430.296} C_VEL
LIN {X 0,Y 593.143,Z 330.343,A -85,B 0,C 180,E1 28427.242,E2 28427.242} C_VEL
LIN {X 0,Y 593.188,Z 330.307,A -85,B 0,C 180,E1 28424.052,E2 28424.052} C_VEL
LIN {X 0,Y 593.15,Z 330.32,A -85,B 0,C 180,E1 28421.013,E2 28421.013} C_VEL
LIN {X 0,Y 593.179,Z 330.339,A -85,B 0,C 180,E1 28417.711,E2 28417.711} C_VEL
LIN {X 0,Y 593.176,Z 330.302,A -85,B 0,C 180,E1 28414.542,E2 28414.542} C_VEL
LIN {X 0,Y 593.161,Z 330.317,A -85,B 0,C 180,E1 28411.287,E2 28411.287} C_VEL
LIN {X 0,Y 593.173,Z 330.426,A -85,B 0,C 180,E1 28408.811,E2 28408.811} C_VEL
LIN {X 0,Y 594.477,Z 333.788,A -85,B 0,C 180,E1 28408.234,E2 28408.234} C_VEL
LIN {X 0,Y 595.75,Z 335.487,A -85,B 0,C 180,E1 28407.856,E2 28407.856} C_VEL
LIN {X 0,Y 597.578,Z 339.331,A -85,B 0,C 180,E1 28407.171,E2 28407.171} C_VEL
LIN {X 0,Y 601.176,Z 346.396,A -85,B 0,C 180,E1 28405.92,E2 28405.92} C_VEL
LIN {X 0,Y 608.664,Z 356.576,A -85,B 0,C 180,E1 28404.672,E2 28404.672} C_VEL
LIN {X 0,Y 618.564,Z 370.164,A -85,B 0,C 180,E1 28403.151,E2 28403.151} C_VEL
LIN {X 0,Y 630.61,Z 387.596,A -85,B 0,C 180,E1 28401.414,E2 28401.414} C_VEL
LIN {X 0,Y 640.304,Z 402.28,A -85,B 0,C 180,E1 28400.096,E2 28400.096} C_VEL
LIN {X 0,Y 635.022,Z 609.008,A -85,B 0,C 180,E1 28397.195,E2 28397.195} C_VEL
LIN {X 0,Y 629.815,Z 823.672,A -85,B 0,C 180,E1 28394.243,E2 28394.243} C_VEL
LIN {X 0,Y 628.772,Z 845.512,A -85,B 0,C 180,E1 28393.869,E2 28393.869} C_VEL
LIN {X 0,Y 627.428,Z 867.206,A -85,B 0,C 180,E1 28393.388,E2 28393.388} C_VEL
LIN {X 0,Y 625.53,Z 892.603,A -85,B 0,C 180,E1 28392.678,E2 28392.678} C_VEL
LIN {X 0,Y 623.1,Z 918.73,A -85,B 0,C 180,E1 28391.754,E2 28391.754} C_VEL
LIN {X 0,Y 620.977,Z 939.461,A -85,B 0,C 180,E1 28390.883,E2 28390.883} C_VEL
LIN {X 0,Y 618.823,Z 958.689,A -85,B 0,C 180,E1 28389.96,E2 28389.96} C_VEL
LIN {X 0,Y 616.543,Z 977.638,A -85,B 0,C 180,E1 28388.933,E2 28388.933} C_VEL
LIN {X 0,Y 614.088,Z 997.061,A -85,B 0,C 180,E1 28387.749,E2 28387.749} C_VEL
LIN {X 0,Y 610.965,Z 1020.891,A -85,B 0,C 180,E1 28386.096,E2 28386.096} C_VEL
LIN {X 0,Y 608.093,Z 1041.618,A -85,B 0,C 180,E1 28384.445,E2 28384.445} C_VEL
LIN {X 0,Y 605.719,Z 1059.054,A -85,B 0,C 180,E1 28382.893,E2 28382.893} C_VEL
LIN {X 0,Y 603.289,Z 1077.267,A -85,B 0,C 180,E1 28381.092,E2 28381.092} C_VEL
LIN {X 0,Y 600.702,Z 1097.147,A -85,B 0,C 180,E1 28378.862,E2 28378.862} C_VEL
LIN {X 0,Y 598.746,Z 1112.645,A -85,B 0,C 180,E1 28376.903,E2 28376.903} C_VEL
LIN {X 0,Y 597.074,Z 1127.45,A -85,B 0,C 180,E1 28374.815,E2 28374.815} C_VEL
LIN {X 0,Y 595.364,Z 1143.704,A -85,B 0,C 180,E1 28372.201,E2 28372.201} C_VEL
LIN {X 0,Y 594.298,Z 1155.271,A -85,B 0,C 180,E1 28370.073,E2 28370.073} C_VEL
LIN {X 0,Y 593.5,Z 1165.449,A -85,B 0,C 180,E1 28367.957,E2 28367.957} C_VEL
LIN {X 0,Y 592.788,Z 1176.306,A -85,B 0,C 180,E1 28365.356,E2 28365.356} C_VEL
LIN {X 0,Y 592.348,Z 1185.18,A -85,B 0,C 180,E1 28362.775,E2 28362.775} C_VEL
LIN {X 0,Y 592.108,Z 1191.86,A -85,B 0,C 180,E1 28360.41,E2 28360.41} C_VEL
LIN {X 0,Y 591.981,Z 1197.542,A -85,B 0,C 180,E1 28357.863,E2 28357.863} C_VEL
LIN {X 0,Y 591.927,Z 1201.661,A -85,B 0,C 180,E1 28355.233,E2 28355.233} C_VEL
LIN {X 0,Y 591.915,Z 1203.925,A -85,B 0,C 180,E1 28352.905,E2 28352.905} C_VEL
LIN {X 0,Y 591.895,Z 1204.849,A -85,B 0,C 180,E1 28350.678,E2 28350.678} C_VEL
LIN {X 0,Y 591.908,Z 1204.623,A -85,B 0,C 180,E1 28348.354,E2 28348.354} C_VEL
LIN {X 0,Y 591.918,Z 1202.789,A -85,B 0,C 180,E1 28345.738,E2 28345.738} C_VEL
LIN {X 0,Y 591.945,Z 1199.546,A -85,B 0,C 180,E1 28343.307,E2 28343.307} C_VEL
LIN {X 0,Y 592.022,Z 1195.103,A -85,B 0,C 180,E1 28340.963,E2 28340.963} C_VEL
LIN {X 0,Y 592.224,Z 1188.471,A -85,B 0,C 180,E1 28338.31,E2 28338.31} C_VEL
LIN {X 0,Y 592.556,Z 1180.571,A -85,B 0,C 180,E1 28335.838,E2 28335.838} C_VEL
LIN {X 0,Y 593.029,Z 1172.305,A -85,B 0,C 180,E1 28333.646,E2 28333.646} C_VEL
LIN {X 0,Y 593.709,Z 1162.694,A -85,B 0,C 180,E1 28331.44,E2 28331.44} C_VEL
LIN {X 0,Y 594.841,Z 1149.447,A -85,B 0,C 180,E1 28328.815,E2 28328.815} C_VEL
LIN {X 0,Y 596.107,Z 1136.315,A -85,B 0,C 180,E1 28326.567,E2 28326.567} C_VEL
LIN {X 0,Y 597.54,Z 1122.985,A -85,B 0,C 180,E1 28324.53,E2 28324.53} C_VEL
LIN {X 0,Y 599.573,Z 1106.413,A -85,B 0,C 180,E1 28322.273,E2 28322.273} C_VEL
LIN {X 0,Y 601.819,Z 1088.229,A -85,B 0,C 180,E1 28320.105,E2 28320.105} C_VEL
LIN {X 0,Y 603.941,Z 1072.291,A -85,B 0,C 180,E1 28318.4,E2 28318.4} C_VEL
LIN {X 0,Y 606.351,Z 1054.613,A -85,B 0,C 180,E1 28316.694,E2 28316.694} C_VEL
LIN {X 0,Y 609.496,Z 1031.566,A -85,B 0,C 180,E1 28314.729,E2 28314.729} C_VEL
LIN {X 0,Y 612.158,Z 1011.517,A -85,B 0,C 180,E1 28313.229,E2 28313.229} C_VEL
LIN {X 0,Y 614.692,Z 992.1,A -85,B 0,C 180,E1 28311.934,E2 28311.934} C_VEL
LIN {X 0,Y 617.675,Z 968.572,A -85,B 0,C 180,E1 28310.549,E2 28310.549} C_VEL
LIN {X 0,Y 620.469,Z 943.986,A -85,B 0,C 180,E1 28309.32,E2 28309.32} C_VEL
LIN {X 0,Y 622.709,Z 922.583,A -85,B 0,C 180,E1 28308.399,E2 28308.399} C_VEL
LIN {X 0,Y 624.662,Z 901.901,A -85,B 0,C 180,E1 28307.634,E2 28307.634} C_VEL
LIN {X 0,Y 626.528,Z 879.601,A -85,B 0,C 180,E1 28306.939,E2 28306.939} C_VEL
LIN {X 0,Y 628.488,Z 851.06,A -85,B 0,C 180,E1 28306.24,E2 28306.24} C_VEL
LIN {X 0,Y 629.695,Z 826.788,A -85,B 0,C 180,E1 28305.804,E2 28305.804} C_VEL
LIN {X 0,Y 633.823,Z 658.219,A -85,B 0,C 180,E1 28303.485,E2 28303.485} C_VEL
LIN {X 0,Y 639.251,Z 442.299,A -85,B 0,C 180,E1 28300.472,E2 28300.472} C_VEL
LIN {X 0,Y 640.217,Z 402.034,A -85,B 0,C 180,E1 28299.89,E2 28299.89} C_VEL
LIN {X 0,Y 624.589,Z 378.681,A -85,B 0,C 180,E1 28297.733,E2 28297.733} C_VEL
LIN {X 0,Y 610.845,Z 359.365,A -85,B 0,C 180,E1 28295.672,E2 28295.672} C_VEL
LIN {X 0,Y 601.148,Z 346.339,A -85,B 0,C 180,E1 28294.076,E2 28294.076} C_VEL
LIN {X 0,Y 599.793,Z 343.618,A -85,B 0,C 180,E1 28293.605,E2 28293.605} C_VEL
LIN {X 0,Y 597.556,Z 339.302,A -85,B 0,C 180,E1 28292.83,E2 28292.83} C_VEL
LIN {X 0,Y 595.737,Z 335.437,A -85,B 0,C 180,E1 28292.145,E2 28292.145} C_VEL
LIN {X 0,Y 593.439,Z 331.617,A -85,B 0,C 180,E1 28291.375,E2 28291.375} C_VEL
LIN {X 0,Y 593.16,Z 330.325,A -85,B 0,C 180,E1 28291.166,E2 28291.166} C_VEL
LIN {X 0,Y 593.201,Z 330.333,A -85,B 0,C 180,E1 28287.967,E2 28287.967} C_VEL
LIN {X 0,Y 593.151,Z 330.305,A -85,B 0,C 180,E1 28284.819,E2 28284.819} C_VEL
LIN {X 0,Y 593.198,Z 330.318,A -85,B 0,C 180,E1 28281.663,E2 28281.663} C_VEL
LIN {X 0,Y 593.156,Z 330.334,A -85,B 0,C 180,E1 28278.477,E2 28278.477} C_VEL
LIN {X 0,Y 593.173,Z 330.299,A -85,B 0,C 180,E1 28275.246,E2 28275.246} C_VEL
LIN {X 0,Y 593.161,Z 330.342,A -85,B 0,C 180,E1 28272.164,E2 28272.164} C_VEL
LIN {X 0,Y 593.145,Z 330.301,A -85,B 0,C 180,E1 28268.824,E2 28268.824} C_VEL
LIN {X 0,Y 593.176,Z 330.342,A -85,B 0,C 180,E1 28265.805,E2 28265.805} C_VEL
LIN {X 0,Y 593.136,Z 330.303,A -85,B 0,C 180,E1 28262.609,E2 28262.609} C_VEL
LIN {X 0,Y 593.177,Z 330.343,A -85,B 0,C 180,E1 28259.614,E2 28259.614} C_VEL
LIN {X 0,Y 593.128,Z 330.305,A -85,B 0,C 180,E1 28256.424,E2 28256.424} C_VEL
LIN {X 0,Y 593.178,Z 330.342,A -85,B 0,C 180,E1 28253.418,E2 28253.418} C_VEL
LIN {X 0,Y 593.124,Z 330.307,A -85,B 0,C 180,E1 28250.295,E2 28250.295} C_VEL
LIN {X 0,Y 593.163,Z 330.341,A -85,B 0,C 180,E1 28247.341,E2 28247.341} C_VEL
LIN {X 0,Y 593.118,Z 330.313,A -85,B 0,C 180,E1 28244.151,E2 28244.151} C_VEL
LIN {X 0,Y 593.154,Z 330.329,A -85,B 0,C 180,E1 28241.218,E2 28241.218} C_VEL
LIN {X 0,Y 593.114,Z 330.329,A -85,B 0,C 180,E1 28237.999,E2 28237.999} C_VEL
LIN {X 0,Y 593.133,Z 330.314,A -85,B 0,C 180,E1 28235.181,E2 28235.181} C_VEL
LIN {X 0,Y 593.115,Z 330.351,A -85,B 0,C 180,E1 28231.943,E2 28231.943} C_VEL
LIN {X 0,Y 593.114,Z 330.31,A -85,B 0,C 180,E1 28229.17,E2 28229.17} C_VEL
LIN {X 0,Y 593.169,Z 330.542,A -85,B 0,C 180,E1 28226.874,E2 28226.874} C_VEL
LIN {X 0,Y 594.263,Z 333.478,A -85,B 0,C 180,E1 28226.648,E2 28226.648} C_VEL
LIN {X 0,Y 596.874,Z 336.135,A -85,B 0,C 180,E1 28226.208,E2 28226.208} C_VEL
LIN {X 0,Y 597.884,Z 337.09,A -85,B 0,C 180,E1 28226.042,E2 28226.042} C_VEL
LIN {X 0,Y 600.296,Z 340.803,A -85,B 0,C 180,E1 28225.621,E2 28225.621} C_VEL
LIN {X 0,Y 602.738,Z 343.136,A -85,B 0,C 180,E1 28225.232,E2 28225.232} C_VEL
LIN {X 0,Y 605.879,Z 347.339,A -85,B 0,C 180,E1 28224.717,E2 28224.717} C_VEL
LIN {X 0,Y 607.544,Z 349.396,A -85,B 0,C 180,E1 28224.452,E2 28224.452} C_VEL
LIN {X 0,Y 611.316,Z 353.883,A -85,B 0,C 180,E1 28223.868,E2 28223.868} C_VEL
LIN {X 0,Y 624.604,Z 371.334,A -85,B 0,C 180,E1 28221.893,E2 28221.893} C_VEL
LIN {X 0,Y 635.369,Z 385.948,A -85,B 0,C 180,E1 28220.405,E2 28220.405} C_VEL
LIN {X 0,Y 640.038,Z 392.799,A -85,B 0,C 180,E1 28219.78,E2 28219.78} C_VEL
LIN {X 0,Y 635.561,Z 563.903,A -85,B 0,C 180,E1 28217.372,E2 28217.372} C_VEL
LIN {X 0,Y 634.688,Z 571.608,A -85,B 0,C 180,E1 28217.331,E2 28217.331} C_VEL
LIN {X 0,Y 629.92,Z 592.266,A -85,B 0,C 180,E1 28217.464,E2 28217.464} C_VEL
LIN {X 0,Y 629.244,Z 598.874,A -85,B 0,C 180,E1 28217.422,E2 28217.422} C_VEL
LIN {X 0,Y 624.009,Z 797.217,A -85,B 0,C 180,E1 28214.664,E2 28214.664} C_VEL
LIN {X 0,Y 622.774,Z 820.824,A -85,B 0,C 180,E1 28214.238,E2 28214.238} C_VEL
LIN {X 0,Y 620.706,Z 849.438,A -85,B 0,C 180,E1 28213.535,E2 28213.535} C_VEL
LIN {X 0,Y 618.813,Z 870.973,A -85,B 0,C 180,E1 28212.862,E2 28212.862} C_VEL
LIN {X 0,Y 616.734,Z 891.657,A -85,B 0,C 180,E1 28212.096,E2 28212.096} C_VEL
LIN {X 0,Y 614.514,Z 912.031,A -85,B 0,C 180,E1 28211.221,E2 28211.221} C_VEL
LIN {X 0,Y 612.147,Z 931.973,A -85,B 0,C 180,E1 28210.24,E2 28210.24} C_VEL
LIN {X 0,Y 609.113,Z 955.819,A -85,B 0,C 180,E1 28208.899,E2 28208.899} C_VEL
LIN {X 0,Y 605.899,Z 978.755,A -85,B 0,C 180,E1 28207.393,E2 28207.393} C_VEL
LIN {X 0,Y 603.259,Z 997.349,A -85,B 0,C 180,E1 28206.016,E2 28206.016} C_VEL
LIN {X 0,Y 600.58,Z 1016.006,A -85,B 0,C 180,E1 28204.474,E2 28204.474} C_VEL
LIN {X 0,Y 597.409,Z 1038.341,A -85,B 0,C 180,E1 28202.382,E2 28202.382} C_VEL
LIN {X 0,Y 594.953,Z 1055.541,A -85,B 0,C 180,E1 28200.555,E2 28200.555} C_VEL
LIN {X 0,Y 592.803,Z 1071.026,A -85,B 0,C 180,E1 28198.731,E2 28198.731} C_VEL
LIN {X 0,Y 590.598,Z 1088.443,A -85,B 0,C 180,E1 28196.439,E2 28196.439} C_VEL
LIN {X 0,Y 588.667,Z 1104.198,A -85,B 0,C 180,E1 28194.057,E2 28194.057} C_VEL
LIN {X 0,Y 587.36,Z 1116.333,A -85,B 0,C 180,E1 28191.994,E2 28191.994} C_VEL
LIN {X 0,Y 586.216,Z 1128.653,A -85,B 0,C 180,E1 28189.634,E2 28189.634} C_VEL
LIN {X 0,Y 585.239,Z 1140.497,A -85,B 0,C 180,E1 28186.986,E2 28186.986} C_VEL
LIN {X 0,Y 584.709,Z 1149.001,A -85,B 0,C 180,E1 28184.761,E2 28184.761} C_VEL
LIN {X 0,Y 584.328,Z 1156.252,A -85,B 0,C 180,E1 28182.551,E2 28182.551} C_VEL
LIN {X 0,Y 584.096,Z 1162.998,A -85,B 0,C 180,E1 28180.056,E2 28180.056} C_VEL
LIN {X 0,Y 583.968,Z 1168.512,A -85,B 0,C 180,E1 28177.378,E2 28177.378} C_VEL
LIN {X 0,Y 583.924,Z 1171.946,A -85,B 0,C 180,E1 28175.01,E2 28175.01} C_VEL
LIN {X 0,Y 583.909,Z 1174.094,A -85,B 0,C 180,E1 28172.65,E2 28172.65} C_VEL
LIN {X 0,Y 583.915,Z 1174.996,A -85,B 0,C 180,E1 28170,E2 28170} C_VEL
LIN {X 0,Y 583.907,Z 1174.157,A -85,B 0,C 180,E1 28167.35,E2 28167.35} C_VEL
LIN {X 0,Y 583.921,Z 1172.051,A -85,B 0,C 180,E1 28164.99,E2 28164.99} C_VEL
LIN {X 0,Y 583.967,Z 1168.658,A -85,B 0,C 180,E1 28162.622,E2 28162.622} C_VEL
LIN {X 0,Y 584.089,Z 1163.218,A -85,B 0,C 180,E1 28159.944,E2 28159.944} C_VEL
LIN {X 0,Y 584.321,Z 1156.524,A -85,B 0,C 180,E1 28157.449,E2 28157.449} C_VEL
LIN {X 0,Y 584.687,Z 1149.316,A -85,B 0,C 180,E1 28155.238,E2 28155.238} C_VEL
LIN {X 0,Y 585.215,Z 1140.857,A -85,B 0,C 180,E1 28153.013,E2 28153.013} C_VEL
LIN {X 0,Y 586.179,Z 1129.096,A -85,B 0,C 180,E1 28150.365,E2 28150.365} C_VEL
LIN {X 0,Y 587.308,Z 1116.819,A -85,B 0,C 180,E1 28148.004,E2 28148.004} C_VEL
LIN {X 0,Y 588.602,Z 1104.733,A -85,B 0,C 180,E1 28145.94,E2 28145.94} C_VEL
LIN {X 0,Y 590.422,Z 1089.746,A -85,B 0,C 180,E1 28143.661,E2 28143.661} C_VEL
LIN {X 0,Y 592.642,Z 1072.192,A -85,B 0,C 180,E1 28141.323,E2 28141.323} C_VEL
LIN {X 0,Y 594.772,Z 1056.748,A -85,B 0,C 180,E1 28139.49,E2 28139.49} C_VEL
LIN {X 0,Y 597.135,Z 1040.157,A -85,B 0,C 180,E1 28137.714,E2 28137.714} C_VEL
LIN {X 0,Y 600.225,Z 1018.777,A -85,B 0,C 180,E1 28135.676,E2 28135.676} C_VEL
LIN {X 0,Y 603.045,Z 998.865,A -85,B 0,C 180,E1 28134.012,E2 28134.012} C_VEL
LIN {X 0,Y 605.636,Z 980.611,A -85,B 0,C 180,E1 28132.648,E2 28132.648} C_VEL
LIN {X 0,Y 608.371,Z 960.787,A -85,B 0,C 180,E1 28131.324,E2 28131.324} C_VEL
LIN {X 0,Y 611.729,Z 935.453,A -85,B 0,C 180,E1 28129.849,E2 28129.849} C_VEL
LIN {X 0,Y 614.332,Z 913.594,A -85,B 0,C 180,E1 28128.76,E2 28128.76} C_VEL
LIN {X 0,Y 616.539,Z 893.503,A -85,B 0,C 180,E1 28127.888,E2 28127.888} C_VEL
LIN {X 0,Y 618.602,Z 873.068,A -85,B 0,C 180,E1 28127.12,E2 28127.12} C_VEL
LIN {X 0,Y 620.482,Z 852.051,A -85,B 0,C 180,E1 28126.452,E2 28126.452} C_VEL
LIN {X 0,Y 622.364,Z 827.443,A -85,B 0,C 180,E1 28125.814,E2 28125.814} C_VEL
LIN {X 0,Y 623.921,Z 799.365,A -85,B 0,C 180,E1 28125.278,E2 28125.278} C_VEL
LIN {X 0,Y 625.884,Z 729.202,A -85,B 0,C 180,E1 28124.295,E2 28124.295} C_VEL
LIN {X 0,Y 631.564,Z 511.883,A -85,B 0,C 180,E1 28121.265,E2 28121.265} C_VEL
LIN {X 0,Y 634.654,Z 396.402,A -85,B 0,C 180,E1 28119.609,E2 28119.609} C_VEL
LIN {X 0,Y 622.861,Z 380.07,A -85,B 0,C 180,E1 28117.969,E2 28117.969} C_VEL
LIN {X 0,Y 611.03,Z 364.506,A -85,B 0,C 180,E1 28116.21,E2 28116.21} C_VEL
LIN {X 0,Y 606.617,Z 359.055,A -85,B 0,C 180,E1 28115.523,E2 28115.523} C_VEL
LIN {X 0,Y 602.552,Z 353.856,A -85,B 0,C 180,E1 28114.867,E2 28114.867} C_VEL
LIN {X 0,Y 598.804,Z 349.067,A -85,B 0,C 180,E1 28114.245,E2 28114.245} C_VEL
LIN {X 0,Y 595.453,Z 345.142,A -85,B 0,C 180,E1 28113.681,E2 28113.681} C_VEL
LIN {X 0,Y 594.133,Z 343.271,A -85,B 0,C 180,E1 28113.447,E2 28113.447} C_VEL
LIN {X 0,Y 591.071,Z 339.965,A -85,B 0,C 180,E1 28112.919,E2 28112.919} C_VEL
LIN {X 0,Y 589.829,Z 337.651,A -85,B 0,C 180,E1 28112.679,E2 28112.679} C_VEL
LIN {X 0,Y 586.867,Z 335.366,A -85,B 0,C 180,E1 28112.17,E2 28112.17} C_VEL
LIN {X 0,Y 585.394,Z 332.422,A -85,B 0,C 180,E1 28111.871,E2 28111.871} C_VEL
LIN {X 0,Y 585.183,Z 331.321,A -85,B 0,C 180,E1 28111.809,E2 28111.809} C_VEL
LIN {X 0,Y 585.165,Z 331.328,A -85,B 0,C 180,E1 28108.567,E2 28108.567} C_VEL
LIN {X 0,Y 585.183,Z 331.294,A -85,B 0,C 180,E1 28105.722,E2 28105.722} C_VEL
LIN {X 0,Y 585.176,Z 331.336,A -85,B 0,C 180,E1 28102.504,E2 28102.504} C_VEL
LIN {X 0,Y 585.183,Z 331.294,A -85,B 0,C 180,E1 28099.671,E2 28099.671} C_VEL
LIN {X 0,Y 585.181,Z 331.319,A -85,B 0,C 180,E1 28096.376,E2 28096.376} C_VEL
LIN {X 0,Y 585.19,Z 331.305,A -85,B 0,C 180,E1 28093.538,E2 28093.538} C_VEL
LIN {X 0,Y 585.185,Z 331.309,A -85,B 0,C 180,E1 28090.211,E2 28090.211} C_VEL
LIN {X 0,Y 585.21,Z 331.311,A -85,B 0,C 180,E1 28087.264,E2 28087.264} C_VEL
LIN {X 0,Y 585.188,Z 331.305,A -85,B 0,C 180,E1 28084.017,E2 28084.017} C_VEL
LIN {X 0,Y 585.234,Z 331.311,A -85,B 0,C 180,E1 28080.979,E2 28080.979} C_VEL
LIN {X 0,Y 585.193,Z 331.303,A -85,B 0,C 180,E1 28077.846,E2 28077.846} C_VEL
LIN {X 0,Y 585.251,Z 331.313,A -85,B 0,C 180,E1 28074.706,E2 28074.706} C_VEL
LIN {X 0,Y 585.194,Z 331.295,A -85,B 0,C 180,E1 28071.55,E2 28071.55} C_VEL
LIN {X 0,Y 585.261,Z 331.324,A -85,B 0,C 180,E1 28068.37,E2 28068.37} C_VEL
LIN {X 0,Y 585.201,Z 331.289,A -85,B 0,C 180,E1 28065.251,E2 28065.251} C_VEL
LIN {X 0,Y 585.259,Z 331.326,A -85,B 0,C 180,E1 28062.09,E2 28062.09} C_VEL
LIN {X 0,Y 585.216,Z 331.295,A -85,B 0,C 180,E1 28058.884,E2 28058.884} C_VEL
LIN {X 0,Y 585.231,Z 331.297,A -85,B 0,C 180,E1 28055.577,E2 28055.577} C_VEL
LIN {X 0,Y 585.252,Z 331.332,A -85,B 0,C 180,E1 28052.419,E2 28052.419} C_VEL
LIN {X 0,Y 585.281,Z 331.475,A -85,B 0,C 180,E1 28049.927,E2 28049.927} C_VEL
LIN {X 0,Y 586.486,Z 334.709,A -85,B 0,C 180,E1 28049.352,E2 28049.352} C_VEL
LIN {X 0,Y 587.944,Z 336.91,A -85,B 0,C 180,E1 28048.869,E2 28048.869} C_VEL
LIN {X 0,Y 589.796,Z 340.471,A -85,B 0,C 180,E1 28048.18,E2 28048.18} C_VEL
LIN {X 0,Y 593.155,Z 346.737,A -85,B 0,C 180,E1 28047.039,E2 28047.039} C_VEL
LIN {X 0,Y 605.147,Z 362.783,A -85,B 0,C 180,E1 28045.016,E2 28045.016} C_VEL
LIN {X 0,Y 615.474,Z 377.139,A -85,B 0,C 180,E1 28043.4,E2 28043.4} C_VEL
LIN {X 0,Y 626.905,Z 393.827,A -85,B 0,C 180,E1 28041.724,E2 28041.724} C_VEL
LIN {X 0,Y 635.041,Z 406.225,A -85,B 0,C 180,E1 28040.594,E2 28040.594} C_VEL
LIN {X 0,Y 629.424,Z 614.525,A -85,B 0,C 180,E1 28037.652,E2 28037.652} C_VEL
LIN {X 0,Y 624.02,Z 824.696,A -85,B 0,C 180,E1 28034.739,E2 28034.739} C_VEL
LIN {X 0,Y 622.895,Z 846.713,A -85,B 0,C 180,E1 28034.355,E2 28034.355} C_VEL
LIN {X 0,Y 621.316,Z 870.732,A -85,B 0,C 180,E1 28033.807,E2 28033.807} C_VEL
LIN {X 0,Y 619.043,Z 898.064,A -85,B 0,C 180,E1 28033,E2 28033} C_VEL
LIN {X 0,Y 616.91,Z 919.973,A -85,B 0,C 180,E1 28032.208,E2 28032.208} C_VEL
LIN {X 0,Y 614.683,Z 940.587,A -85,B 0,C 180,E1 28031.331,E2 28031.331} C_VEL
LIN {X 0,Y 612.542,Z 958.685,A -85,B 0,C 180,E1 28030.454,E2 28030.454} C_VEL
LIN {X 0,Y 610.137,Z 977.635,A -85,B 0,C 180,E1 28029.421,E2 28029.421} C_VEL
LIN {X 0,Y 607.445,Z 997.869,A -85,B 0,C 180,E1 28028.176,E2 28028.176} C_VEL
LIN {X 0,Y 603.998,Z 1022.551,A -85,B 0,C 180,E1 28026.433,E2 28026.433} C_VEL
LIN {X 0,Y 601.133,Z 1042.225,A -85,B 0,C 180,E1 28024.844,E2 28024.844} C_VEL
LIN {X 0,Y 598.621,Z 1059.608,A -85,B 0,C 180,E1 28023.277,E2 28023.277} C_VEL
LIN {X 0,Y 595.844,Z 1079.333,A -85,B 0,C 180,E1 28021.295,E2 28021.295} C_VEL
LIN {X 0,Y 593.241,Z 1097.991,A -85,B 0,C 180,E1 28019.149,E2 28019.149} C_VEL
LIN {X 0,Y 591.276,Z 1112.615,A -85,B 0,C 180,E1 28017.275,E2 28017.275} C_VEL
LIN {X 0,Y 589.498,Z 1127.186,A -85,B 0,C 180,E1 28015.197,E2 28015.197} C_VEL
LIN {X 0,Y 587.644,Z 1143.706,A -85,B 0,C 180,E1 28012.509,E2 28012.509} C_VEL
LIN {X 0,Y 586.477,Z 1155.376,A -85,B 0,C 180,E1 28010.33,E2 28010.33} C_VEL
LIN {X 0,Y 585.631,Z 1165.448,A -85,B 0,C 180,E1 28008.206,E2 28008.206} C_VEL
LIN {X 0,Y 584.857,Z 1176.307,A -85,B 0,C 180,E1 28005.569,E2 28005.569} C_VEL
LIN {X 0,Y 584.39,Z 1185.176,A -85,B 0,C 180,E1 28002.952,E2 28002.952} C_VEL
LIN {X 0,Y 584.128,Z 1191.603,A -85,B 0,C 180,E1 28000.653,E2 28000.653} C_VEL
LIN {X 0,Y 583.992,Z 1197.151,A -85,B 0,C 180,E1 27998.17,E2 27998.17} C_VEL
LIN {X 0,Y 583.93,Z 1201.428,A -85,B 0,C 180,E1 27995.502,E2 27995.502} C_VEL
LIN {X 0,Y 583.917,Z 1203.854,A -85,B 0,C 180,E1 27993.043,E2 27993.043} C_VEL
LIN {X 0,Y 583.905,Z 1204.804,A -85,B 0,C 180,E1 27990.883,E2 27990.883} C_VEL
LIN {X 0,Y 583.915,Z 1204.736,A -85,B 0,C 180,E1 27988.823,E2 27988.823} C_VEL
LIN {X 0,Y 583.913,Z 1203.51,A -85,B 0,C 180,E1 27986.466,E2 27986.466} C_VEL
LIN {X 0,Y 583.943,Z 1200.337,A -85,B 0,C 180,E1 27983.709,E2 27983.709} C_VEL
LIN {X 0,Y 584.019,Z 1195.926,A -85,B 0,C 180,E1 27981.236,E2 27981.236} C_VEL
LIN {X 0,Y 584.152,Z 1190.586,A -85,B 0,C 180,E1 27978.948,E2 27978.948} C_VEL
LIN {X 0,Y 584.519,Z 1182.685,A -85,B 0,C 180,E1 27976.245,E2 27976.245} C_VEL
LIN {X 0,Y 585.07,Z 1173.113,A -85,B 0,C 180,E1 27973.622,E2 27973.622} C_VEL
LIN {X 0,Y 585.743,Z 1164.074,A -85,B 0,C 180,E1 27971.488,E2 27971.488} C_VEL
LIN {X 0,Y 586.693,Z 1153.206,A -85,B 0,C 180,E1 27969.239,E2 27969.239} C_VEL
LIN {X 0,Y 588.226,Z 1138.277,A -85,B 0,C 180,E1 27966.563,E2 27966.563} C_VEL
LIN {X 0,Y 589.783,Z 1124.56,A -85,B 0,C 180,E1 27964.413,E2 27964.413} C_VEL
LIN {X 0,Y 591.601,Z 1110.303,A -85,B 0,C 180,E1 27962.414,E2 27962.414} C_VEL
LIN {X 0,Y 594.11,Z 1091.609,A -85,B 0,C 180,E1 27960.083,E2 27960.083} C_VEL
LIN {X 0,Y 596.592,Z 1073.81,A -85,B 0,C 180,E1 27958.135,E2 27958.135} C_VEL
LIN {X 0,Y 598.947,Z 1057.387,A -85,B 0,C 180,E1 27956.515,E2 27956.515} C_VEL
LIN {X 0,Y 601.698,Z 1038.571,A -85,B 0,C 180,E1 27954.845,E2 27954.845} C_VEL
LIN {X 0,Y 605.028,Z 1015.188,A -85,B 0,C 180,E1 27953.02,E2 27953.02} C_VEL
LIN {X 0,Y 607.749,Z 995.427,A -85,B 0,C 180,E1 27951.667,E2 27951.667} C_VEL
LIN {X 0,Y 610.362,Z 975.836,A -85,B 0,C 180,E1 27950.475,E2 27950.475} C_VEL
LIN {X 0,Y 612.906,Z 955.676,A -85,B 0,C 180,E1 27949.39,E2 27949.39} C_VEL
LIN {X 0,Y 615.754,Z 931.539,A -85,B 0,C 180,E1 27948.26,E2 27948.26} C_VEL
LIN {X 0,Y 618.267,Z 906.249,A -85,B 0,C 180,E1 27947.28,E2 27947.28} C_VEL
LIN {X 0,Y 620.181,Z 884.693,A -85,B 0,C 180,E1 27946.583,E2 27946.583} C_VEL
LIN {X 0,Y 621.817,Z 863.409,A -85,B 0,C 180,E1 27946.014,E2 27946.014} C_VEL
LIN {X 0,Y 623.185,Z 841.667,A -85,B 0,C 180,E1 27945.546,E2 27945.546} C_VEL
LIN {X 0,Y 624.45,Z 813.521,A -85,B 0,C 180,E1 27945.094,E2 27945.094} C_VEL
LIN {X 0,Y 630.055,Z 590.308,A -85,B 0,C 180,E1 27942.01,E2 27942.01} C_VEL
LIN {X 0,Y 635.032,Z 406.022,A -85,B 0,C 180,E1 27939.401,E2 27939.401} C_VEL
LIN {X 0,Y 619.961,Z 383.609,A -85,B 0,C 180,E1 27937.273,E2 27937.273} C_VEL
LIN {X 0,Y 609.986,Z 369.459,A -85,B 0,C 180,E1 27935.759,E2 27935.759} C_VEL
LIN {X 0,Y 602.345,Z 359.035,A -85,B 0,C 180,E1 27934.534,E2 27934.534} C_VEL
LIN {X 0,Y 595.286,Z 349.729,A -85,B 0,C 180,E1 27933.345,E2 27933.345} C_VEL
LIN {X 0,Y 592.644,Z 345.672,A -85,B 0,C 180,E1 27932.824,E2 27932.824} C_VEL
LIN {X 0,Y 590.578,Z 341.988,A -85,B 0,C 180,E1 27932.115,E2 27932.115} C_VEL
LIN {X 0,Y 589.149,Z 339.571,A -85,B 0,C 180,E1 27931.63,E2 27931.63} C_VEL
LIN {X 0,Y 587.394,Z 335.866,A -85,B 0,C 180,E1 27930.936,E2 27930.936} C_VEL
LIN {X 0,Y 585.52,Z 332.54,A -85,B 0,C 180,E1 27930.25,E2 27930.25} C_VEL
LIN {X 0,Y 585.255,Z 331.287,A -85,B 0,C 180,E1 27930.039,E2 27930.039} C_VEL
LIN {X 0,Y 585.217,Z 331.321,A -85,B 0,C 180,E1 27926.894,E2 27926.894} C_VEL
LIN {X 0,Y 585.259,Z 331.311,A -85,B 0,C 180,E1 27923.671,E2 27923.671} C_VEL
LIN {X 0,Y 585.212,Z 331.289,A -85,B 0,C 180,E1 27920.565,E2 27920.565} C_VEL
LIN {X 0,Y 585.238,Z 331.33,A -85,B 0,C 180,E1 27917.248,E2 27917.248} C_VEL
LIN {X 0,Y 585.224,Z 331.29,A -85,B 0,C 180,E1 27914.142,E2 27914.142} C_VEL
LIN {X 0,Y 585.209,Z 331.319,A -85,B 0,C 180,E1 27910.833,E2 27910.833} C_VEL
LIN {X 0,Y 585.256,Z 331.303,A -85,B 0,C 180,E1 27907.658,E2 27907.658} C_VEL
LIN {X 0,Y 585.197,Z 331.309,A -85,B 0,C 180,E1 27904.508,E2 27904.508} C_VEL
LIN {X 0,Y 585.26,Z 331.308,A -85,B 0,C 180,E1 27901.371,E2 27901.371} C_VEL
LIN {X 0,Y 585.19,Z 331.307,A -85,B 0,C 180,E1 27898.335,E2 27898.335} C_VEL
LIN {X 0,Y 585.257,Z 331.31,A -85,B 0,C 180,E1 27895.198,E2 27895.198} C_VEL
LIN {X 0,Y 585.185,Z 331.305,A -85,B 0,C 180,E1 27892.143,E2 27892.143} C_VEL
LIN {X 0,Y 585.249,Z 331.316,A -85,B 0,C 180,E1 27888.968,E2 27888.968} C_VEL
LIN {X 0,Y 585.177,Z 331.3,A -85,B 0,C 180,E1 27885.958,E2 27885.958} C_VEL
LIN {X 0,Y 585.253,Z 331.322,A -85,B 0,C 180,E1 27882.911,E2 27882.911} C_VEL
LIN {X 0,Y 585.17,Z 331.293,A -85,B 0,C 180,E1 27879.808,E2 27879.808} C_VEL
LIN {X 0,Y 585.253,Z 331.332,A -85,B 0,C 180,E1 27876.755,E2 27876.755} C_VEL
LIN {X 0,Y 585.166,Z 331.302,A -85,B 0,C 180,E1 27873.623,E2 27873.623} C_VEL
LIN {X 0,Y 585.236,Z 331.297,A -85,B 0,C 180,E1 27870.524,E2 27870.524} C_VEL
LIN {X 0,Y 585.2,Z 331.432,A -85,B 0,C 180,E1 27868.082,E2 27868.082} C_VEL
LIN {X 0,Y 586.239,Z 334.445,A -85,B 0,C 180,E1 27867.849,E2 27867.849} C_VEL
LIN {X 0,Y 588.632,Z 336.989,A -85,B 0,C 180,E1 27867.42,E2 27867.42} C_VEL
LIN {X 0,Y 590.067,Z 338.03,A -85,B 0,C 180,E1 27867.177,E2 27867.177} C_VEL
LIN {X 0,Y 592.458,Z 341.766,A -85,B 0,C 180,E1 27866.735,E2 27866.735} C_VEL
LIN {X 0,Y 594.884,Z 344.148,A -85,B 0,C 180,E1 27866.326,E2 27866.326} C_VEL
LIN {X 0,Y 597.993,Z 348.333,A -85,B 0,C 180,E1 27865.789,E2 27865.789} C_VEL
LIN {X 0,Y 599.889,Z 350.372,A -85,B 0,C 180,E1 27865.479,E2 27865.479} C_VEL
LIN {X 0,Y 605.046,Z 357.086,A -85,B 0,C 180,E1 27864.632,E2 27864.632} C_VEL
LIN {X 0,Y 609.825,Z 363.009,A -85,B 0,C 180,E1 27863.882,E2 27863.882} C_VEL
LIN {X 0,Y 620.68,Z 377.151,A -85,B 0,C 180,E1 27862.254,E2 27862.254} C_VEL
LIN {X 0,Y 632.039,Z 392.746,A -85,B 0,C 180,E1 27860.655,E2 27860.655} C_VEL
LIN {X 0,Y 634.79,Z 396.943,A -85,B 0,C 180,E1 27860.277,E2 27860.277} C_VEL
LIN {X 0,Y 629.244,Z 598.874,A -85,B 0,C 180,E1 27857.422,E2 27857.422} C_VEL
LIN {X 0,Y 628.362,Z 606.58,A -85,B 0,C 180,E1 27857.383,E2 27857.383} C_VEL
LIN {X 0,Y 623.551,Z 627.23,A -85,B 0,C 180,E1 27857.522,E2 27857.522} C_VEL
LIN {X 0,Y 622.889,Z 633.836,A -85,B 0,C 180,E1 27857.478,E2 27857.478} C_VEL
LIN {X 0,Y 618.336,Z 797.662,A -85,B 0,C 180,E1 27855.183,E2 27855.183} C_VEL
LIN {X 0,Y 617.019,Z 821.783,A -85,B 0,C 180,E1 27854.744,E2 27854.744} C_VEL
LIN {X 0,Y 614.856,Z 850.193,A -85,B 0,C 180,E1 27854.038,E2 27854.038} C_VEL
LIN {X 0,Y 612.847,Z 871.992,A -85,B 0,C 180,E1 27853.35,E2 27853.35} C_VEL
LIN {X 0,Y 610.747,Z 891.934,A -85,B 0,C 180,E1 27852.605,E2 27852.605} C_VEL
LIN {X 0,Y 608.465,Z 911.658,A -85,B 0,C 180,E1 27851.75,E2 27851.75} C_VEL
LIN {X 0,Y 605.949,Z 931.572,A -85,B 0,C 180,E1 27850.764,E2 27850.764} C_VEL
LIN {X 0,Y 602.822,Z 955.065,A -85,B 0,C 180,E1 27849.439,E2 27849.439} C_VEL
LIN {X 0,Y 599.395,Z 978.349,A -85,B 0,C 180,E1 27847.903,E2 27847.903} C_VEL
LIN {X 0,Y 596.594,Z 997.052,A -85,B 0,C 180,E1 27846.51,E2 27846.51} C_VEL
LIN {X 0,Y 593.797,Z 1015.404,A -85,B 0,C 180,E1 27844.984,E2 27844.984} C_VEL
LIN {X 0,Y 590.575,Z 1036.824,A -85,B 0,C 180,E1 27842.977,E2 27842.977} C_VEL
LIN {X 0,Y 587.809,Z 1055.082,A -85,B 0,C 180,E1 27841.024,E2 27841.024} C_VEL
LIN {X 0,Y 585.589,Z 1070.185,A -85,B 0,C 180,E1 27839.231,E2 27839.231} C_VEL
LIN {X 0,Y 583.409,Z 1085.679,A -85,B 0,C 180,E1 27837.189,E2 27837.189} C_VEL
LIN {X 0,Y 581.197,Z 1102.931,A -85,B 0,C 180,E1 27834.603,E2 27834.603} C_VEL
LIN {X 0,Y 579.698,Z 1115.778,A -85,B 0,C 180,E1 27832.404,E2 27832.404} C_VEL
LIN {X 0,Y 578.526,Z 1127.219,A -85,B 0,C 180,E1 27830.2,E2 27830.2} C_VEL
LIN {X 0,Y 577.422,Z 1139.73,A -85,B 0,C 180,E1 27827.419,E2 27827.419} C_VEL
LIN {X 0,Y 576.8,Z 1148.649,A -85,B 0,C 180,E1 27825.071,E2 27825.071} C_VEL
LIN {X 0,Y 576.392,Z 1155.948,A -85,B 0,C 180,E1 27822.829,E2 27822.829} C_VEL
LIN {X 0,Y 576.122,Z 1162.755,A -85,B 0,C 180,E1 27820.297,E2 27820.297} C_VEL
LIN {X 0,Y 575.972,Z 1168.51,A -85,B 0,C 180,E1 27817.481,E2 27817.481} C_VEL
LIN {X 0,Y 575.925,Z 1171.944,A -85,B 0,C 180,E1 27815.08,E2 27815.08} C_VEL
LIN {X 0,Y 575.911,Z 1174.024,A -85,B 0,C 180,E1 27812.786,E2 27812.786} C_VEL
LIN {X 0,Y 575.894,Z 1174.906,A -85,B 0,C 180,E1 27810.398,E2 27810.398} C_VEL
LIN {X 0,Y 575.909,Z 1174.351,A -85,B 0,C 180,E1 27807.612,E2 27807.612} C_VEL
LIN {X 0,Y 575.919,Z 1172.274,A -85,B 0,C 180,E1 27805.12,E2 27805.12} C_VEL
LIN {X 0,Y 575.962,Z 1169.133,A -85,B 0,C 180,E1 27802.82,E2 27802.82} C_VEL
LIN {X 0,Y 576.069,Z 1164.355,A -85,B 0,C 180,E1 27800.308,E2 27800.308} C_VEL
LIN {X 0,Y 576.315,Z 1157.429,A -85,B 0,C 180,E1 27797.577,E2 27797.577} C_VEL
LIN {X 0,Y 576.709,Z 1150.019,A -85,B 0,C 180,E1 27795.235,E2 27795.235} C_VEL
LIN {X 0,Y 577.231,Z 1142.073,A -85,B 0,C 180,E1 27793.082,E2 27793.082} C_VEL
LIN {X 0,Y 577.982,Z 1132.89,A -85,B 0,C 180,E1 27790.916,E2 27790.916} C_VEL
LIN {X 0,Y 579.232,Z 1120.254,A -85,B 0,C 180,E1 27788.321,E2 27788.321} C_VEL
LIN {X 0,Y 580.785,Z 1106.207,A -85,B 0,C 180,E1 27785.848,E2 27785.848} C_VEL
LIN {X 0,Y 582.408,Z 1093.269,A -85,B 0,C 180,E1 27783.819,E2 27783.819} C_VEL
LIN {X 0,Y 584.677,Z 1076.732,A -85,B 0,C 180,E1 27781.503,E2 27781.503} C_VEL
LIN {X 0,Y 587.272,Z 1058.593,A -85,B 0,C 180,E1 27779.285,E2 27779.285} C_VEL
LIN {X 0,Y 589.639,Z 1042.813,A -85,B 0,C 180,E1 27777.556,E2 27777.556} C_VEL
LIN {X 0,Y 592.189,Z 1026.15,A -85,B 0,C 180,E1 27775.906,E2 27775.906} C_VEL
LIN {X 0,Y 595.444,Z 1005.082,A -85,B 0,C 180,E1 27774.037,E2 27774.037} C_VEL
LIN {X 0,Y 598.726,Z 982.803,A -85,B 0,C 180,E1 27772.323,E2 27772.323} C_VEL
LIN {X 0,Y 601.519,Z 963.593,A -85,B 0,C 180,E1 27771.013,E2 27771.013} C_VEL
LIN {X 0,Y 604.288,Z 943.783,A -85,B 0,C 180,E1 27769.812,E2 27769.812} C_VEL
LIN {X 0,Y 607.668,Z 918.239,A -85,B 0,C 180,E1 27768.464,E2 27768.464} C_VEL
LIN {X 0,Y 610.407,Z 895.011,A -85,B 0,C 180,E1 27767.429,E2 27767.429} C_VEL
LIN {X 0,Y 612.633,Z 874.05,A -85,B 0,C 180,E1 27766.631,E2 27766.631} C_VEL
LIN {X 0,Y 614.586,Z 853.234,A -85,B 0,C 180,E1 27765.962,E2 27765.962} C_VEL
LIN {X 0,Y 616.39,Z 830.796,A -85,B 0,C 180,E1 27765.37,E2 27765.37} C_VEL
LIN {X 0,Y 618.139,Z 802.469,A -85,B 0,C 180,E1 27764.801,E2 27764.801} C_VEL
LIN {X 0,Y 619.695,Z 753.018,A -85,B 0,C 180,E1 27764.093,E2 27764.093} C_VEL
LIN {X 0,Y 625.795,Z 530.115,A -85,B 0,C 180,E1 27760.97,E2 27760.97} C_VEL
LIN {X 0,Y 629.567,Z 400.673,A -85,B 0,C 180,E1 27759.118,E2 27759.118} C_VEL
LIN {X 0,Y 618.264,Z 385.055,A -85,B 0,C 180,E1 27757.51,E2 27757.51} C_VEL
LIN {X 0,Y 607.351,Z 370.607,A -85,B 0,C 180,E1 27755.851,E2 27755.851} C_VEL
LIN {X 0,Y 599.083,Z 360.171,A -85,B 0,C 180,E1 27754.516,E2 27754.516} C_VEL
LIN {X 0,Y 595.615,Z 355.759,A -85,B 0,C 180,E1 27753.931,E2 27753.931} C_VEL
LIN {X 0,Y 592.074,Z 351.343,A -85,B 0,C 180,E1 27753.318,E2 27753.318} C_VEL
LIN {X 0,Y 587.628,Z 345.981,A -85,B 0,C 180,E1 27752.527,E2 27752.527} C_VEL
LIN {X 0,Y 586.698,Z 344.657,A -85,B 0,C 180,E1 27752.354,E2 27752.354} C_VEL
LIN {X 0,Y 583.582,Z 341.626,A -85,B 0,C 180,E1 27751.794,E2 27751.794} C_VEL
LIN {X 0,Y 581.82,Z 338.541,A -85,B 0,C 180,E1 27751.439,E2 27751.439} C_VEL
LIN {X 0,Y 578.851,Z 336.197,A -85,B 0,C 180,E1 27750.895,E2 27750.895} C_VEL
LIN {X 0,Y 577.433,Z 333.389,A -85,B 0,C 180,E1 27750.589,E2 27750.589} C_VEL
LIN {X 0,Y 577.213,Z 332.286,A -85,B 0,C 180,E1 27750.501,E2 27750.501} C_VEL
LIN {X 0,Y 577.275,Z 332.318,A -85,B 0,C 180,E1 27747.527,E2 27747.527} C_VEL
LIN {X 0,Y 577.224,Z 332.298,A -85,B 0,C 180,E1 27744.339,E2 27744.339} C_VEL
LIN {X 0,Y 577.27,Z 332.286,A -85,B 0,C 180,E1 27741.437,E2 27741.437} C_VEL
LIN {X 0,Y 577.236,Z 332.321,A -85,B 0,C 180,E1 27738.272,E2 27738.272} C_VEL
LIN {X 0,Y 577.281,Z 332.274,A -85,B 0,C 180,E1 27735.263,E2 27735.263} C_VEL
LIN {X 0,Y 577.242,Z 332.326,A -85,B 0,C 180,E1 27732.099,E2 27732.099} C_VEL
LIN {X 0,Y 577.304,Z 332.268,A -85,B 0,C 180,E1 27728.968,E2 27728.968} C_VEL
LIN {X 0,Y 577.246,Z 332.325,A -85,B 0,C 180,E1 27725.866,E2 27725.866} C_VEL
LIN {X 0,Y 577.309,Z 332.266,A -85,B 0,C 180,E1 27722.68,E2 27722.68} C_VEL
LIN {X 0,Y 577.252,Z 332.325,A -85,B 0,C 180,E1 27719.603,E2 27719.603} C_VEL
LIN {X 0,Y 577.305,Z 332.267,A -85,B 0,C 180,E1 27716.425,E2 27716.425} C_VEL
LIN {X 0,Y 577.262,Z 332.324,A -85,B 0,C 180,E1 27713.336,E2 27713.336} C_VEL
LIN {X 0,Y 577.298,Z 332.273,A -85,B 0,C 180,E1 27710.127,E2 27710.127} C_VEL
LIN {X 0,Y 577.271,Z 332.312,A -85,B 0,C 180,E1 27707.089,E2 27707.089} C_VEL
LIN {X 0,Y 577.28,Z 332.293,A -85,B 0,C 180,E1 27703.704,E2 27703.704} C_VEL
LIN {X 0,Y 577.302,Z 332.279,A -85,B 0,C 180,E1 27700.577,E2 27700.577} C_VEL
LIN {X 0,Y 577.276,Z 332.324,A -85,B 0,C 180,E1 27697.278,E2 27697.278} C_VEL
LIN {X 0,Y 577.318,Z 332.277,A -85,B 0,C 180,E1 27694.122,E2 27694.122} C_VEL
LIN {X 0,Y 577.28,Z 332.306,A -85,B 0,C 180,E1 27691.159,E2 27691.159} C_VEL
LIN {X 0,Y 578.352,Z 335.38,A -85,B 0,C 180,E1 27690.594,E2 27690.594} C_VEL
LIN {X 0,Y 580.073,Z 337.846,A -85,B 0,C 180,E1 27690.008,E2 27690.008} C_VEL
LIN {X 0,Y 581.796,Z 341.384,A -85,B 0,C 180,E1 27689.307,E2 27689.307} C_VEL
LIN {X 0,Y 582.844,Z 343.359,A -85,B 0,C 180,E1 27688.91,E2 27688.91} C_VEL
LIN {X 0,Y 584.596,Z 346.345,A -85,B 0,C 180,E1 27688.354,E2 27688.354} C_VEL
LIN {X 0,Y 589.314,Z 352.333,A -85,B 0,C 180,E1 27687.491,E2 27687.491} C_VEL
LIN {X 0,Y 602.201,Z 369.78,A -85,B 0,C 180,E1 27685.272,E2 27685.272} C_VEL
LIN {X 0,Y 614.317,Z 386.779,A -85,B 0,C 180,E1 27683.36,E2 27683.36} C_VEL
LIN {X 0,Y 629.828,Z 409.986,A -85,B 0,C 180,E1 27681.104,E2 27681.104} C_VEL
LIN {X 0,Y 623.923,Z 617.868,A -85,B 0,C 180,E1 27678.148,E2 27678.148} C_VEL
LIN {X 0,Y 618.308,Z 824.861,A -85,B 0,C 180,E1 27675.258,E2 27675.258} C_VEL
LIN {X 0,Y 617.109,Z 847.1,A -85,B 0,C 180,E1 27674.866,E2 27674.866} C_VEL
LIN {X 0,Y 615.295,Z 873.471,A -85,B 0,C 180,E1 27674.254,E2 27674.254} C_VEL
LIN {X 0,Y 612.944,Z 899.358,A -85,B 0,C 180,E1 27673.467,E2 27673.467} C_VEL
LIN {X 0,Y 610.759,Z 920.66,A -85,B 0,C 180,E1 27672.686,E2 27672.686} C_VEL
LIN {X 0,Y 608.549,Z 940.471,A -85,B 0,C 180,E1 27671.841,E2 27671.841} C_VEL
LIN {X 0,Y 606.269,Z 958.983,A -85,B 0,C 180,E1 27670.943,E2 27670.943} C_VEL
LIN {X 0,Y 603.66,Z 978.532,A -85,B 0,C 180,E1 27669.866,E2 27669.866} C_VEL
LIN {X 0,Y 600.518,Z 1001.112,A -85,B 0,C 180,E1 27668.453,E2 27668.453} C_VEL
LIN {X 0,Y 597.051,Z 1024.224,A -85,B 0,C 180,E1 27666.776,E2 27666.776} C_VEL
LIN {X 0,Y 594.203,Z 1042.831,A -85,B 0,C 180,E1 27665.251,E2 27665.251} C_VEL
LIN {X 0,Y 591.55,Z 1060.162,A -85,B 0,C 180,E1 27663.669,E2 27663.669} C_VEL
LIN {X 0,Y 588.525,Z 1080.343,A -85,B 0,C 180,E1 27661.609,E2 27661.609} C_VEL
LIN {X 0,Y 585.85,Z 1098.461,A -85,B 0,C 180,E1 27659.49,E2 27659.49} C_VEL
LIN {X 0,Y 583.724,Z 1113.383,A -85,B 0,C 180,E1 27657.547,E2 27657.547} C_VEL
LIN {X 0,Y 581.679,Z 1129.285,A -85,B 0,C 180,E1 27655.232,E2 27655.232} C_VEL
LIN {X 0,Y 579.852,Z 1144.405,A -85,B 0,C 180,E1 27652.698,E2 27652.698} C_VEL
LIN {X 0,Y 578.642,Z 1155.782,A -85,B 0,C 180,E1 27650.534,E2 27650.534} C_VEL
LIN {X 0,Y 577.699,Z 1166.364,A -85,B 0,C 180,E1 27648.256,E2 27648.256} C_VEL
LIN {X 0,Y 576.865,Z 1177.39,A -85,B 0,C 180,E1 27645.479,E2 27645.479} C_VEL
LIN {X 0,Y 576.432,Z 1185.173,A -85,B 0,C 180,E1 27643.134,E2 27643.134} C_VEL
LIN {X 0,Y 576.142,Z 1191.612,A -85,B 0,C 180,E1 27640.798,E2 27640.798} C_VEL
LIN {X 0,Y 575.999,Z 1197.151,A -85,B 0,C 180,E1 27638.284,E2 27638.284} C_VEL
LIN {X 0,Y 575.932,Z 1201.427,A -85,B 0,C 180,E1 27635.579,E2 27635.579} C_VEL
LIN {X 0,Y 575.917,Z 1203.851,A -85,B 0,C 180,E1 27633.085,E2 27633.085} C_VEL
LIN {X 0,Y 575.905,Z 1204.804,A -85,B 0,C 180,E1 27630.895,E2 27630.895} C_VEL
LIN {X 0,Y 575.915,Z 1204.736,A -85,B 0,C 180,E1 27628.806,E2 27628.806} C_VEL
LIN {X 0,Y 575.913,Z 1203.51,A -85,B 0,C 180,E1 27626.417,E2 27626.417} C_VEL
LIN {X 0,Y 575.946,Z 1200.337,A -85,B 0,C 180,E1 27623.621,E2 27623.621} C_VEL
LIN {X 0,Y 576.025,Z 1195.923,A -85,B 0,C 180,E1 27621.113,E2 27621.113} C_VEL
LIN {X 0,Y 576.176,Z 1190.583,A -85,B 0,C 180,E1 27618.793,E2 27618.793} C_VEL
LIN {X 0,Y 576.569,Z 1182.685,A -85,B 0,C 180,E1 27616.052,E2 27616.052} C_VEL
LIN {X 0,Y 577.161,Z 1173.112,A -85,B 0,C 180,E1 27613.391,E2 27613.391} C_VEL
LIN {X 0,Y 577.893,Z 1164.073,A -85,B 0,C 180,E1 27611.227,E2 27611.227} C_VEL
LIN {X 0,Y 578.925,Z 1153.208,A -85,B 0,C 180,E1 27608.947,E2 27608.947} C_VEL
LIN {X 0,Y 580.564,Z 1138.275,A -85,B 0,C 180,E1 27606.234,E2 27606.234} C_VEL
LIN {X 0,Y 582.162,Z 1125.083,A -85,B 0,C 180,E1 27604.136,E2 27604.136} C_VEL
LIN {X 0,Y 584.064,Z 1111.071,A -85,B 0,C 180,E1 27602.138,E2 27602.138} C_VEL
LIN {X 0,Y 586.669,Z 1092.855,A -85,B 0,C 180,E1 27599.817,E2 27599.817} C_VEL
LIN {X 0,Y 589.384,Z 1074.495,A -85,B 0,C 180,E1 27597.776,E2 27597.776} C_VEL
LIN {X 0,Y 591.895,Z 1057.941,A -85,B 0,C 180,E1 27596.12,E2 27596.12} C_VEL
LIN {X 0,Y 594.593,Z 1040.394,A -85,B 0,C 180,E1 27594.539,E2 27594.539} C_VEL
LIN {X 0,Y 598.029,Z 1017.907,A -85,B 0,C 180,E1 27592.737,E2 27592.737} C_VEL
LIN {X 0,Y 601.141,Z 996.316,A -85,B 0,C 180,E1 27591.234,E2 27591.234} C_VEL
LIN {X 0,Y 603.894,Z 976.732,A -85,B 0,C 180,E1 27590.029,E2 27590.029} C_VEL
LIN {X 0,Y 606.433,Z 957.683,A -85,B 0,C 180,E1 27588.989,E2 27588.989} C_VEL
LIN {X 0,Y 608.764,Z 938.682,A -85,B 0,C 180,E1 27588.078,E2 27588.078} C_VEL
LIN {X 0,Y 611.147,Z 917.159,A -85,B 0,C 180,E1 27587.174,E2 27587.174} C_VEL
LIN {X 0,Y 613.92,Z 889.004,A -85,B 0,C 180,E1 27586.198,E2 27586.198} C_VEL
LIN {X 0,Y 615.83,Z 865.63,A -85,B 0,C 180,E1 27585.551,E2 27585.551} C_VEL
LIN {X 0,Y 617.28,Z 844.172,A -85,B 0,C 180,E1 27585.076,E2 27585.076} C_VEL
LIN {X 0,Y 618.435,Z 821.844,A -85,B 0,C 180,E1 27584.697,E2 27584.697} C_VEL
LIN {X 0,Y 624.321,Z 603.3,A -85,B 0,C 180,E1 27581.647,E2 27581.647} C_VEL
LIN {X 0,Y 629.807,Z 409.958,A -85,B 0,C 180,E1 27578.894,E2 27578.894} C_VEL
LIN {X 0,Y 613.83,Z 386.066,A -85,B 0,C 180,E1 27576.569,E2 27576.569} C_VEL
LIN {X 0,Y 600.132,Z 366.832,A -85,B 0,C 180,E1 27574.39,E2 27574.39} C_VEL
LIN {X 0,Y 588.785,Z 351.813,A -85,B 0,C 180,E1 27572.427,E2 27572.427} C_VEL
LIN {X 0,Y 583.843,Z 345.386,A -85,B 0,C 180,E1 27571.49,E2 27571.49} C_VEL
LIN {X 0,Y 582.081,Z 341.736,A -85,B 0,C 180,E1 27570.791,E2 27570.791} C_VEL
LIN {X 0,Y 580.237,Z 338.386,A -85,B 0,C 180,E1 27570.097,E2 27570.097} C_VEL
LIN {X 0,Y 579.494,Z 336.834,A -85,B 0,C 180,E1 27569.788,E2 27569.788} C_VEL
LIN {X 0,Y 577.629,Z 333.827,A -85,B 0,C 180,E1 27569.106,E2 27569.106} C_VEL
LIN {X 0,Y 577.279,Z 332.287,A -85,B 0,C 180,E1 27568.841,E2 27568.841} C_VEL
LIN {X 0,Y 577.313,Z 332.274,A -85,B 0,C 180,E1 27565.658,E2 27565.658} C_VEL
LIN {X 0,Y 577.294,Z 332.321,A -85,B 0,C 180,E1 27562.399,E2 27562.399} C_VEL
LIN {X 0,Y 577.276,Z 332.29,A -85,B 0,C 180,E1 27559.004,E2 27559.004} C_VEL
LIN {X 0,Y 577.314,Z 332.28,A -85,B 0,C 180,E1 27555.882,E2 27555.882} C_VEL
LIN {X 0,Y 577.269,Z 332.316,A -85,B 0,C 180,E1 27552.708,E2 27552.708} C_VEL
LIN {X 0,Y 577.317,Z 332.269,A -85,B 0,C 180,E1 27549.571,E2 27549.571} C_VEL
LIN {X 0,Y 577.262,Z 332.324,A -85,B 0,C 180,E1 27546.465,E2 27546.465} C_VEL
LIN {X 0,Y 577.311,Z 332.267,A -85,B 0,C 180,E1 27543.277,E2 27543.277} C_VEL
LIN {X 0,Y 577.259,Z 332.324,A -85,B 0,C 180,E1 27540.198,E2 27540.198} C_VEL
LIN {X 0,Y 577.299,Z 332.268,A -85,B 0,C 180,E1 27537.022,E2 27537.022} C_VEL
LIN {X 0,Y 577.257,Z 332.324,A -85,B 0,C 180,E1 27533.935,E2 27533.935} C_VEL
LIN {X 0,Y 577.267,Z 332.274,A -85,B 0,C 180,E1 27530.629,E2 27530.629} C_VEL
LIN {X 0,Y 577.262,Z 332.325,A -85,B 0,C 180,E1 27527.597,E2 27527.597} C_VEL
LIN {X 0,Y 577.248,Z 332.282,A -85,B 0,C 180,E1 27524.323,E2 27524.323} C_VEL
LIN {X 0,Y 577.258,Z 332.313,A -85,B 0,C 180,E1 27521.415,E2 27521.415} C_VEL
LIN {X 0,Y 577.242,Z 332.298,A -85,B 0,C 180,E1 27518.135,E2 27518.135} C_VEL
LIN {X 0,Y 577.243,Z 332.292,A -85,B 0,C 180,E1 27515.326,E2 27515.326} C_VEL
LIN {X 0,Y 577.24,Z 332.33,A -85,B 0,C 180,E1 27512.003,E2 27512.003} C_VEL
LIN {X 0,Y 577.242,Z 332.406,A -85,B 0,C 180,E1 27509.363,E2 27509.363} C_VEL
LIN {X 0,Y 578.239,Z 335.277,A -85,B 0,C 180,E1 27509.127,E2 27509.127} C_VEL
LIN {X 0,Y 580.66,Z 337.86,A -85,B 0,C 180,E1 27508.665,E2 27508.665} C_VEL
LIN {X 0,Y 582.161,Z 338.985,A -85,B 0,C 180,E1 27508.394,E2 27508.394} C_VEL
LIN {X 0,Y 584.454,Z 342.732,A -85,B 0,C 180,E1 27507.942,E2 27507.942} C_VEL
LIN {X 0,Y 587.308,Z 345.403,A -85,B 0,C 180,E1 27507.435,E2 27507.435} C_VEL
LIN {X 0,Y 590.436,Z 349.535,A -85,B 0,C 180,E1 27506.868,E2 27506.868} C_VEL
LIN {X 0,Y 592.145,Z 351.464,A -85,B 0,C 180,E1 27506.571,E2 27506.571} C_VEL
LIN {X 0,Y 595.825,Z 355.949,A -85,B 0,C 180,E1 27505.938,E2 27505.938} C_VEL
LIN {X 0,Y 602.438,Z 364.504,A -85,B 0,C 180,E1 27504.835,E2 27504.835} C_VEL
LIN {X 0,Y 609.142,Z 372.854,A -85,B 0,C 180,E1 27503.777,E2 27503.777} C_VEL
LIN {X 0,Y 621.476,Z 389.434,A -85,B 0,C 180,E1 27501.931,E2 27501.931} C_VEL
LIN {X 0,Y 629.594,Z 400.879,A -85,B 0,C 180,E1 27500.785,E2 27500.785} C_VEL
LIN {X 0,Y 623.143,Z 624.601,A -85,B 0,C 180,E1 27497.608,E2 27497.608} C_VEL
LIN {X 0,Y 622.889,Z 633.836,A -85,B 0,C 180,E1 27497.478,E2 27497.478} C_VEL
LIN {X 0,Y 622.036,Z 641.537,A -85,B 0,C 180,E1 27497.435,E2 27497.435} C_VEL
LIN {X 0,Y 617.218,Z 662.184,A -85,B 0,C 180,E1 27497.577,E2 27497.577} C_VEL
LIN {X 0,Y 616.515,Z 668.796,A -85,B 0,C 180,E1 27497.537,E2 27497.537} C_VEL
LIN {X 0,Y 612.71,Z 798.23,A -85,B 0,C 180,E1 27495.71,E2 27495.71} C_VEL
LIN {X 0,Y 611.286,Z 823.21,A -85,B 0,C 180,E1 27495.25,E2 27495.25} C_VEL
LIN {X 0,Y 609.058,Z 850.923,A -85,B 0,C 180,E1 27494.551,E2 27494.551} C_VEL
LIN {X 0,Y 607.005,Z 872.276,A -85,B 0,C 180,E1 27493.873,E2 27493.873} C_VEL
LIN {X 0,Y 604.81,Z 892.216,A -85,B 0,C 180,E1 27493.125,E2 27493.125} C_VEL
LIN {X 0,Y 602.365,Z 912.436,A -85,B 0,C 180,E1 27492.241,E2 27492.241} C_VEL
LIN {X 0,Y 599.779,Z 931.835,A -85,B 0,C 180,E1 27491.272,E2 27491.272} C_VEL
LIN {X 0,Y 596.341,Z 955.915,A -85,B 0,C 180,E1 27489.89,E2 27489.89} C_VEL
LIN {X 0,Y 592.806,Z 978.768,A -85,B 0,C 180,E1 27488.366,E2 27488.366} C_VEL
LIN {X 0,Y 589.929,Z 997.058,A -85,B 0,C 180,E1 27486.99,E2 27486.99} C_VEL
LIN {X 0,Y 587.066,Z 1014.869,A -85,B 0,C 180,E1 27485.498,E2 27485.498} C_VEL
LIN {X 0,Y 583.806,Z 1035.282,A -85,B 0,C 180,E1 27483.586,E2 27483.586} C_VEL
LIN {X 0,Y 580.746,Z 1054.31,A -85,B 0,C 180,E1 27481.541,E2 27481.541} C_VEL
LIN {X 0,Y 578.409,Z 1069.343,A -85,B 0,C 180,E1 27479.743,E2 27479.743} C_VEL
LIN {X 0,Y 576.229,Z 1083.842,A -85,B 0,C 180,E1 27477.824,E2 27477.824} C_VEL
LIN {X 0,Y 573.965,Z 1100.36,A -85,B 0,C 180,E1 27475.375,E2 27475.375} C_VEL
LIN {X 0,Y 572.123,Z 1114.696,A -85,B 0,C 180,E1 27472.922,E2 27472.922} C_VEL
LIN {X 0,Y 570.831,Z 1126.136,A -85,B 0,C 180,E1 27470.71,E2 27470.71} C_VEL
LIN {X 0,Y 569.772,Z 1137.101,A -85,B 0,C 180,E1 27468.304,E2 27468.304} C_VEL
LIN {X 0,Y 568.907,Z 1147.941,A -85,B 0,C 180,E1 27465.494,E2 27465.494} C_VEL
LIN {X 0,Y 568.453,Z 1155.644,A -85,B 0,C 180,E1 27463.115,E2 27463.115} C_VEL
LIN {X 0,Y 568.148,Z 1162.249,A -85,B 0,C 180,E1 27460.649,E2 27460.649} C_VEL
LIN {X 0,Y 567.993,Z 1168.003,A -85,B 0,C 180,E1 27457.892,E2 27457.892} C_VEL
LIN {X 0,Y 567.926,Z 1171.828,A -85,B 0,C 180,E1 27455.253,E2 27455.253} C_VEL
LIN {X 0,Y 567.912,Z 1173.953,A -85,B 0,C 180,E1 27452.927,E2 27452.927} C_VEL
LIN {X 0,Y 567.895,Z 1174.862,A -85,B 0,C 180,E1 27450.605,E2 27450.605} C_VEL
LIN {X 0,Y 567.913,Z 1174.565,A -85,B 0,C 180,E1 27447.982,E2 27447.982} C_VEL
LIN {X 0,Y 567.916,Z 1172.612,A -85,B 0,C 180,E1 27445.355,E2 27445.355} C_VEL
LIN {X 0,Y 567.956,Z 1169.449,A -85,B 0,C 180,E1 27442.921,E2 27442.921} C_VEL
LIN {X 0,Y 568.056,Z 1165.185,A -85,B 0,C 180,E1 27440.579,E2 27440.579} C_VEL
LIN {X 0,Y 568.29,Z 1158.874,A -85,B 0,C 180,E1 27437.915,E2 27437.915} C_VEL
LIN {X 0,Y 568.704,Z 1151.076,A -85,B 0,C 180,E1 27435.335,E2 27435.335} C_VEL
LIN {X 0,Y 569.276,Z 1142.88,A -85,B 0,C 180,E1 27433.049,E2 27433.049} C_VEL
LIN {X 0,Y 570.059,Z 1133.803,A -85,B 0,C 180,E1 27430.853,E2 27430.853} C_VEL
LIN {X 0,Y 571.194,Z 1122.9,A -85,B 0,C 180,E1 27428.54,E2 27428.54} C_VEL
LIN {X 0,Y 572.944,Z 1107.896,A -85,B 0,C 180,E1 27425.789,E2 27425.789} C_VEL
LIN {X 0,Y 574.715,Z 1094.496,A -85,B 0,C 180,E1 27423.637,E2 27423.637} C_VEL
LIN {X 0,Y 576.719,Z 1080.606,A -85,B 0,C 180,E1 27421.639,E2 27421.639} C_VEL
LIN {X 0,Y 579.496,Z 1062.29,A -85,B 0,C 180,E1 27419.289,E2 27419.289} C_VEL
LIN {X 0,Y 582.35,Z 1044.197,A -85,B 0,C 180,E1 27417.26,E2 27417.26} C_VEL
LIN {X 0,Y 584.905,Z 1028.353,A -85,B 0,C 180,E1 27415.658,E2 27415.658} C_VEL
LIN {X 0,Y 587.532,Z 1012.068,A -85,B 0,C 180,E1 27414.168,E2 27414.168} C_VEL
LIN {X 0,Y 590.543,Z 993.379,A -85,B 0,C 180,E1 27412.629,E2 27412.629} C_VEL
LIN {X 0,Y 594.346,Z 968.858,A -85,B 0,C 180,E1 27410.856,E2 27410.856} C_VEL
LIN {X 0,Y 597.511,Z 947.452,A -85,B 0,C 180,E1 27409.514,E2 27409.514} C_VEL
LIN {X 0,Y 600.287,Z 927.967,A -85,B 0,C 180,E1 27408.434,E2 27408.434} C_VEL
LIN {X 0,Y 603.029,Z 907.272,A -85,B 0,C 180,E1 27407.43,E2 27407.43} C_VEL
LIN {X 0,Y 606.06,Z 881.652,A -85,B 0,C 180,E1 27406.369,E2 27406.369} C_VEL
LIN {X 0,Y 608.492,Z 857.188,A -85,B 0,C 180,E1 27405.547,E2 27405.547} C_VEL
LIN {X 0,Y 610.318,Z 835.836,A -85,B 0,C 180,E1 27404.958,E2 27404.958} C_VEL
LIN {X 0,Y 611.781,Z 814.859,A -85,B 0,C 180,E1 27404.492,E2 27404.492} C_VEL
LIN {X 0,Y 612.988,Z 791.9,A -85,B 0,C 180,E1 27404.102,E2 27404.102} C_VEL
LIN {X 0,Y 619.449,Z 568.078,A -85,B 0,C 180,E1 27400.949,E2 27400.949} C_VEL
LIN {X 0,Y 624.364,Z 404.792,A -85,B 0,C 180,E1 27398.598,E2 27398.598} C_VEL
LIN {X 0,Y 612.135,Z 387.803,A -85,B 0,C 180,E1 27396.803,E2 27396.803} C_VEL
LIN {X 0,Y 601.028,Z 373.247,A -85,B 0,C 180,E1 27395.056,E2 27395.056} C_VEL
LIN {X 0,Y 592.448,Z 362.414,A -85,B 0,C 180,E1 27393.613,E2 27393.613} C_VEL
LIN {X 0,Y 587.614,Z 356.488,A -85,B 0,C 180,E1 27392.76,E2 27392.76} C_VEL
LIN {X 0,Y 583.604,Z 351.498,A -85,B 0,C 180,E1 27392.024,E2 27392.024} C_VEL
LIN {X 0,Y 580.326,Z 347.857,A -85,B 0,C 180,E1 27391.413,E2 27391.413} C_VEL
LIN {X 0,Y 579.005,Z 345.691,A -85,B 0,C 180,E1 27391.145,E2 27391.145} C_VEL
LIN {X 0,Y 575.864,Z 342.772,A -85,B 0,C 180,E1 27390.55,E2 27390.55} C_VEL
LIN {X 0,Y 574.07,Z 339.64,A -85,B 0,C 180,E1 27390.166,E2 27390.166} C_VEL
LIN {X 0,Y 571.093,Z 337.376,A -85,B 0,C 180,E1 27389.587,E2 27389.587} C_VEL
LIN {X 0,Y 569.537,Z 334.258,A -85,B 0,C 180,E1 27389.228,E2 27389.228} C_VEL
LIN {X 0,Y 569.339,Z 333.278,A -85,B 0,C 180,E1 27389.14,E2 27389.14} C_VEL
LIN {X 0,Y 569.281,Z 333.275,A -85,B 0,C 180,E1 27386.159,E2 27386.159} C_VEL
LIN {X 0,Y 569.341,Z 333.314,A -85,B 0,C 180,E1 27382.947,E2 27382.947} C_VEL
LIN {X 0,Y 569.29,Z 333.266,A -85,B 0,C 180,E1 27379.922,E2 27379.922} C_VEL
LIN {X 0,Y 569.325,Z 333.299,A -85,B 0,C 180,E1 27376.635,E2 27376.635} C_VEL
LIN {X 0,Y 569.3,Z 333.275,A -85,B 0,C 180,E1 27373.716,E2 27373.716} C_VEL
LIN {X 0,Y 569.323,Z 333.286,A -85,B 0,C 180,E1 27370.422,E2 27370.422} C_VEL
LIN {X 0,Y 569.316,Z 333.28,A -85,B 0,C 180,E1 27367.468,E2 27367.468} C_VEL
LIN {X 0,Y 569.316,Z 333.28,A -85,B 0,C 180,E1 27364.129,E2 27364.129} C_VEL
LIN {X 0,Y 569.353,Z 333.287,A -85,B 0,C 180,E1 27361.006,E2 27361.006} C_VEL
LIN {X 0,Y 569.313,Z 333.274,A -85,B 0,C 180,E1 27357.786,E2 27357.786} C_VEL
LIN {X 0,Y 569.381,Z 333.291,A -85,B 0,C 180,E1 27354.558,E2 27354.558} C_VEL
LIN {X 0,Y 569.318,Z 333.266,A -85,B 0,C 180,E1 27351.401,E2 27351.401} C_VEL
LIN {X 0,Y 569.371,Z 333.308,A -85,B 0,C 180,E1 27348.143,E2 27348.143} C_VEL
LIN {X 0,Y 569.333,Z 333.261,A -85,B 0,C 180,E1 27344.995,E2 27344.995} C_VEL
LIN {X 0,Y 569.34,Z 333.298,A -85,B 0,C 180,E1 27341.571,E2 27341.571} C_VEL
LIN {X 0,Y 569.38,Z 333.276,A -85,B 0,C 180,E1 27338.359,E2 27338.359} C_VEL
LIN {X 0,Y 569.334,Z 333.267,A -85,B 0,C 180,E1 27335.181,E2 27335.181} C_VEL
LIN {X 0,Y 569.394,Z 333.455,A -85,B 0,C 180,E1 27332.411,E2 27332.411} C_VEL
LIN {X 0,Y 570.632,Z 336.687,A -85,B 0,C 180,E1 27331.764,E2 27331.764} C_VEL
LIN {X 0,Y 572.069,Z 338.546,A -85,B 0,C 180,E1 27331.271,E2 27331.271} C_VEL
LIN {X 0,Y 573.656,Z 342.042,A -85,B 0,C 180,E1 27330.559,E2 27330.559} C_VEL
LIN {X 0,Y 574.794,Z 343.693,A -85,B 0,C 180,E1 27330.164,E2 27330.164} C_VEL
LIN {X 0,Y 575.85,Z 345.924,A -85,B 0,C 180,E1 27329.794,E2 27329.794} C_VEL
LIN {X 0,Y 583.148,Z 355.151,A -85,B 0,C 180,E1 27328.382,E2 27328.382} C_VEL
LIN {X 0,Y 588.198,Z 361.815,A -85,B 0,C 180,E1 27327.45,E2 27327.45} C_VEL
LIN {X 0,Y 598.059,Z 374.993,A -85,B 0,C 180,E1 27325.736,E2 27325.736} C_VEL
LIN {X 0,Y 610.767,Z 393.06,A -85,B 0,C 180,E1 27323.685,E2 27323.685} C_VEL
LIN {X 0,Y 624.665,Z 414.052,A -85,B 0,C 180,E1 27321.617,E2 27321.617} C_VEL
LIN {X 0,Y 618.346,Z 625.698,A -85,B 0,C 180,E1 27318.59,E2 27318.59} C_VEL
LIN {X 0,Y 612.62,Z 825.674,A -85,B 0,C 180,E1 27315.776,E2 27315.776} C_VEL
LIN {X 0,Y 611.272,Z 849.278,A -85,B 0,C 180,E1 27315.351,E2 27315.351} C_VEL
LIN {X 0,Y 609.019,Z 878.269,A -85,B 0,C 180,E1 27314.641,E2 27314.641} C_VEL
LIN {X 0,Y 606.903,Z 900.497,A -85,B 0,C 180,E1 27313.948,E2 27313.948} C_VEL
LIN {X 0,Y 604.649,Z 921.352,A -85,B 0,C 180,E1 27313.175,E2 27313.175} C_VEL
LIN {X 0,Y 602.301,Z 941.34,A -85,B 0,C 180,E1 27312.311,E2 27312.311} C_VEL
LIN {X 0,Y 599.698,Z 961.485,A -85,B 0,C 180,E1 27311.318,E2 27311.318} C_VEL
LIN {X 0,Y 596.377,Z 985.689,A -85,B 0,C 180,E1 27309.95,E2 27309.95} C_VEL
LIN {X 0,Y 592.841,Z 1008.58,A -85,B 0,C 180,E1 27308.425,E2 27308.425} C_VEL
LIN {X 0,Y 589.919,Z 1027.143,A -85,B 0,C 180,E1 27307.029,E2 27307.029} C_VEL
LIN {X 0,Y 587.055,Z 1044.954,A -85,B 0,C 180,E1 27305.536,E2 27305.536} C_VEL
LIN {X 0,Y 583.745,Z 1065.691,A -85,B 0,C 180,E1 27303.59,E2 27303.59} C_VEL
LIN {X 0,Y 580.656,Z 1084.828,A -85,B 0,C 180,E1 27301.527,E2 27301.527} C_VEL
LIN {X 0,Y 578.359,Z 1099.677,A -85,B 0,C 180,E1 27299.746,E2 27299.746} C_VEL
LIN {X 0,Y 576.184,Z 1114.151,A -85,B 0,C 180,E1 27297.827,E2 27297.827} C_VEL
LIN {X 0,Y 573.927,Z 1130.621,A -85,B 0,C 180,E1 27295.376,E2 27295.376} C_VEL
LIN {X 0,Y 572.08,Z 1144.992,A -85,B 0,C 180,E1 27292.912,E2 27292.912} C_VEL
LIN {X 0,Y 570.805,Z 1156.295,A -85,B 0,C 180,E1 27290.722,E2 27290.722} C_VEL
LIN {X 0,Y 569.731,Z 1167.739,A -85,B 0,C 180,E1 27288.203,E2 27288.203} C_VEL
LIN {X 0,Y 568.894,Z 1178.097,A -85,B 0,C 180,E1 27285.495,E2 27285.495} C_VEL
LIN {X 0,Y 568.461,Z 1185.473,A -85,B 0,C 180,E1 27283.218,E2 27283.218} C_VEL
LIN {X 0,Y 568.153,Z 1191.851,A -85,B 0,C 180,E1 27280.854,E2 27280.854} C_VEL
LIN {X 0,Y 567.998,Z 1197.542,A -85,B 0,C 180,E1 27278.197,E2 27278.197} C_VEL
LIN {X 0,Y 567.93,Z 1201.652,A -85,B 0,C 180,E1 27275.455,E2 27275.455} C_VEL
LIN {X 0,Y 567.916,Z 1203.916,A -85,B 0,C 180,E1 27273.028,E2 27273.028} C_VEL
LIN {X 0,Y 567.901,Z 1204.827,A -85,B 0,C 180,E1 27270.807,E2 27270.807} C_VEL
LIN {X 0,Y 567.913,Z 1204.691,A -85,B 0,C 180,E1 27268.588,E2 27268.588} C_VEL
LIN {X 0,Y 567.916,Z 1203.193,A -85,B 0,C 180,E1 27265.962,E2 27265.962} C_VEL
LIN {X 0,Y 567.949,Z 1200.016,A -85,B 0,C 180,E1 27263.328,E2 27263.328} C_VEL
LIN {X 0,Y 568.035,Z 1195.817,A -85,B 0,C 180,E1 27260.936,E2 27260.936} C_VEL
LIN {X 0,Y 568.22,Z 1190.325,A -85,B 0,C 180,E1 27258.531,E2 27258.531} C_VEL
LIN {X 0,Y 568.638,Z 1182.334,A -85,B 0,C 180,E1 27255.749,E2 27255.749} C_VEL
LIN {X 0,Y 569.259,Z 1173.111,A -85,B 0,C 180,E1 27253.154,E2 27253.154} C_VEL
LIN {X 0,Y 570.047,Z 1164.071,A -85,B 0,C 180,E1 27250.959,E2 27250.959} C_VEL
LIN {X 0,Y 571.169,Z 1153.188,A -85,B 0,C 180,E1 27248.643,E2 27248.643} C_VEL
LIN {X 0,Y 572.909,Z 1138.256,A -85,B 0,C 180,E1 27245.894,E2 27245.894} C_VEL
LIN {X 0,Y 574.631,Z 1125.081,A -85,B 0,C 180,E1 27243.771,E2 27243.771} C_VEL
LIN {X 0,Y 576.655,Z 1111.05,A -85,B 0,C 180,E1 27241.745,E2 27241.745} C_VEL
LIN {X 0,Y 579.417,Z 1092.853,A -85,B 0,C 180,E1 27239.399,E2 27239.399} C_VEL
LIN {X 0,Y 582.254,Z 1074.821,A -85,B 0,C 180,E1 27237.37,E2 27237.37} C_VEL
LIN {X 0,Y 584.874,Z 1058.495,A -85,B 0,C 180,E1 27235.717,E2 27235.717} C_VEL
LIN {X 0,Y 587.607,Z 1041.608,A -85,B 0,C 180,E1 27234.173,E2 27234.173} C_VEL
LIN {X 0,Y 590.732,Z 1022.209,A -85,B 0,C 180,E1 27232.581,E2 27232.581} C_VEL
LIN {X 0,Y 594.466,Z 997.953,A -85,B 0,C 180,E1 27230.842,E2 27230.842} C_VEL
LIN {X 0,Y 597.331,Z 978.472,A -85,B 0,C 180,E1 27229.625,E2 27229.625} C_VEL
LIN {X 0,Y 600.083,Z 958.45,A -85,B 0,C 180,E1 27228.524,E2 27228.524} C_VEL
LIN {X 0,Y 602.541,Z 939.41,A -85,B 0,C 180,E1 27227.601,E2 27227.601} C_VEL
LIN {X 0,Y 604.863,Z 919.477,A -85,B 0,C 180,E1 27226.75,E2 27226.75} C_VEL
LIN {X 0,Y 607.503,Z 894.856,A -85,B 0,C 180,E1 27225.858,E2 27225.858} C_VEL
LIN {X 0,Y 609.921,Z 867.402,A -85,B 0,C 180,E1 27225.068,E2 27225.068} C_VEL
LIN {X 0,Y 611.522,Z 845.047,A -85,B 0,C 180,E1 27224.564,E2 27224.564} C_VEL
LIN {X 0,Y 612.732,Z 823.097,A -85,B 0,C 180,E1 27224.185,E2 27224.185} C_VEL
LIN {X 0,Y 618.823,Z 608.925,A -85,B 0,C 180,E1 27221.173,E2 27221.173} C_VEL
LIN {X 0,Y 624.642,Z 414.028,A -85,B 0,C 180,E1 27218.381,E2 27218.381} C_VEL
LIN {X 0,Y 610.231,Z 392.282,A -85,B 0,C 180,E1 27216.236,E2 27216.236} C_VEL
LIN {X 0,Y 596.917,Z 373.41,A -85,B 0,C 180,E1 27214.078,E2 27214.078} C_VEL
LIN {X 0,Y 585.798,Z 358.574,A -85,B 0,C 180,E1 27212.12,E2 27212.12} C_VEL
LIN {X 0,Y 580.4,Z 351.685,A -85,B 0,C 180,E1 27211.11,E2 27211.11} C_VEL
LIN {X 0,Y 575.143,Z 344.718,A -85,B 0,C 180,E1 27210.032,E2 27210.032} C_VEL
LIN {X 0,Y 574.227,Z 342.748,A -85,B 0,C 180,E1 27209.639,E2 27209.639} C_VEL
LIN {X 0,Y 572.204,Z 339.079,A -85,B 0,C 180,E1 27208.835,E2 27208.835} C_VEL
LIN {X 0,Y 571.448,Z 337.751,A -85,B 0,C 180,E1 27208.534,E2 27208.534} C_VEL
LIN {X 0,Y 569.633,Z 334.527,A -85,B 0,C 180,E1 27207.791,E2 27207.791} C_VEL
LIN {X 0,Y 569.372,Z 333.31,A -85,B 0,C 180,E1 27207.525,E2 27207.525} C_VEL
LIN {X 0,Y 569.366,Z 333.27,A -85,B 0,C 180,E1 27204.264,E2 27204.264} C_VEL
LIN {X 0,Y 569.335,Z 333.268,A -85,B 0,C 180,E1 27200.994,E2 27200.994} C_VEL
LIN {X 0,Y 569.383,Z 333.305,A -85,B 0,C 180,E1 27197.792,E2 27197.792} C_VEL
LIN {X 0,Y 569.323,Z 333.262,A -85,B 0,C 180,E1 27194.546,E2 27194.546} C_VEL
LIN {X 0,Y 569.374,Z 333.299,A -85,B 0,C 180,E1 27191.343,E2 27191.343} C_VEL
LIN {X 0,Y 569.329,Z 333.269,A -85,B 0,C 180,E1 27188.179,E2 27188.179} C_VEL
LIN {X 0,Y 569.335,Z 333.29,A -85,B 0,C 180,E1 27184.836,E2 27184.836} C_VEL
LIN {X 0,Y 569.352,Z 333.277,A -85,B 0,C 180,E1 27181.711,E2 27181.711} C_VEL
LIN {X 0,Y 569.317,Z 333.284,A -85,B 0,C 180,E1 27178.49,E2 27178.49} C_VEL
LIN {X 0,Y 569.377,Z 333.285,A -85,B 0,C 180,E1 27175.266,E2 27175.266} C_VEL
LIN {X 0,Y 569.307,Z 333.277,A -85,B 0,C 180,E1 27172.11,E2 27172.11} C_VEL
LIN {X 0,Y 569.369,Z 333.292,A -85,B 0,C 180,E1 27168.964,E2 27168.964} C_VEL
LIN {X 0,Y 569.3,Z 333.271,A -85,B 0,C 180,E1 27165.869,E2 27165.869} C_VEL
LIN {X 0,Y 569.359,Z 333.304,A -85,B 0,C 180,E1 27162.735,E2 27162.735} C_VEL
LIN {X 0,Y 569.296,Z 333.265,A -85,B 0,C 180,E1 27159.65,E2 27159.65} C_VEL
LIN {X 0,Y 569.332,Z 333.307,A -85,B 0,C 180,E1 27156.395,E2 27156.395} C_VEL
LIN {X 0,Y 569.3,Z 333.278,A -85,B 0,C 180,E1 27153.374,E2 27153.374} C_VEL
LIN {X 0,Y 569.386,Z 333.465,A -85,B 0,C 180,E1 27150.713,E2 27150.713} C_VEL
LIN {X 0,Y 570.492,Z 336.515,A -85,B 0,C 180,E1 27150.437,E2 27150.437} C_VEL
LIN {X 0,Y 572.936,Z 339.035,A -85,B 0,C 180,E1 27149.942,E2 27149.942} C_VEL
LIN {X 0,Y 574.383,Z 340.098,A -85,B 0,C 180,E1 27149.665,E2 27149.665} C_VEL
LIN {X 0,Y 576.707,Z 343.782,A -85,B 0,C 180,E1 27149.18,E2 27149.18} C_VEL
LIN {X 0,Y 579.435,Z 346.323,A -85,B 0,C 180,E1 27148.667,E2 27148.667} C_VEL
LIN {X 0,Y 582.343,Z 350.376,A -85,B 0,C 180,E1 27148.102,E2 27148.102} C_VEL
LIN {X 0,Y 584.612,Z 352.654,A -85,B 0,C 180,E1 27147.691,E2 27147.691} C_VEL
LIN {X 0,Y 588.3,Z 357.137,A -85,B 0,C 180,E1 27147.023,E2 27147.023} C_VEL
LIN {X 0,Y 592.904,Z 362.859,A -85,B 0,C 180,E1 27146.213,E2 27146.213} C_VEL
LIN {X 0,Y 605.983,Z 379.63,A -85,B 0,C 180,E1 27144.055,E2 27144.055} C_VEL
LIN {X 0,Y 617.955,Z 395.827,A -85,B 0,C 180,E1 27142.234,E2 27142.234} C_VEL
LIN {X 0,Y 624.434,Z 405.076,A -85,B 0,C 180,E1 27141.298,E2 27141.298} C_VEL
LIN {X 0,Y 617.714,Z 626.98,A -85,B 0,C 180,E1 27138.127,E2 27138.127} C_VEL
LIN {X 0,Y 616.515,Z 668.796,A -85,B 0,C 180,E1 27137.537,E2 27137.537} C_VEL
LIN {X 0,Y 615.625,Z 676.498,A -85,B 0,C 180,E1 27137.497,E2 27137.497} C_VEL
LIN {X 0,Y 610.815,Z 697.136,A -85,B 0,C 180,E1 27137.641,E2 27137.641} C_VEL
LIN {X 0,Y 610.104,Z 703.745,A -85,B 0,C 180,E1 27137.601,E2 27137.601} C_VEL
LIN {X 0,Y 607.124,Z 799.073,A -85,B 0,C 180,E1 27136.243,E2 27136.243} C_VEL
LIN {X 0,Y 605.508,Z 826.038,A -85,B 0,C 180,E1 27135.736,E2 27135.736} C_VEL
LIN {X 0,Y 603.236,Z 852.382,A -85,B 0,C 180,E1 27135.052,E2 27135.052} C_VEL
LIN {X 0,Y 601.134,Z 873.293,A -85,B 0,C 180,E1 27134.38,E2 27134.38} C_VEL
LIN {X 0,Y 598.773,Z 893.773,A -85,B 0,C 180,E1 27133.602,E2 27133.602} C_VEL
LIN {X 0,Y 596.244,Z 913.727,A -85,B 0,C 180,E1 27132.719,E2 27132.719} C_VEL
LIN {X 0,Y 593.212,Z 935.479,A -85,B 0,C 180,E1 27131.612,E2 27131.612} C_VEL
LIN {X 0,Y 589.381,Z 960.207,A -85,B 0,C 180,E1 27130.139,E2 27130.139} C_VEL
LIN {X 0,Y 586.195,Z 979.607,A -85,B 0,C 180,E1 27128.811,E2 27128.811} C_VEL
LIN {X 0,Y 583.203,Z 997.664,A -85,B 0,C 180,E1 27127.434,E2 27127.434} C_VEL
LIN {X 0,Y 580.304,Z 1014.808,A -85,B 0,C 180,E1 27125.982,E2 27125.982} C_VEL
LIN {X 0,Y 576.846,Z 1035.29,A -85,B 0,C 180,E1 27124.046,E2 27124.046} C_VEL
LIN {X 0,Y 573.543,Z 1054.628,A -85,B 0,C 180,E1 27121.944,E2 27121.944} C_VEL
LIN {X 0,Y 571.072,Z 1069.652,A -85,B 0,C 180,E1 27120.123,E2 27120.123} C_VEL
LIN {X 0,Y 568.705,Z 1084.615,A -85,B 0,C 180,E1 27118.111,E2 27118.111} C_VEL
LIN {X 0,Y 566.21,Z 1101.656,A -85,B 0,C 180,E1 27115.523,E2 27115.523} C_VEL
LIN {X 0,Y 564.358,Z 1115.288,A -85,B 0,C 180,E1 27113.142,E2 27113.142} C_VEL
LIN {X 0,Y 562.998,Z 1126.653,A -85,B 0,C 180,E1 27110.903,E2 27110.903} C_VEL
LIN {X 0,Y 561.803,Z 1138.455,A -85,B 0,C 180,E1 27108.254,E2 27108.254} C_VEL
LIN {X 0,Y 560.959,Z 1148.298,A -85,B 0,C 180,E1 27105.613,E2 27105.613} C_VEL
LIN {X 0,Y 560.494,Z 1155.642,A -85,B 0,C 180,E1 27103.304,E2 27103.304} C_VEL
LIN {X 0,Y 560.17,Z 1161.993,A -85,B 0,C 180,E1 27100.906,E2 27100.906} C_VEL
LIN {X 0,Y 560.009,Z 1167.652,A -85,B 0,C 180,E1 27098.212,E2 27098.212} C_VEL
LIN {X 0,Y 559.932,Z 1171.598,A -85,B 0,C 180,E1 27095.533,E2 27095.533} C_VEL
LIN {X 0,Y 559.913,Z 1173.815,A -85,B 0,C 180,E1 27093.173,E2 27093.173} C_VEL
LIN {X 0,Y 559.905,Z 1174.794,A -85,B 0,C 180,E1 27090.921,E2 27090.921} C_VEL
LIN {X 0,Y 559.907,Z 1174.746,A -85,B 0,C 180,E1 27088.772,E2 27088.772} C_VEL
LIN {X 0,Y 559.913,Z 1173.603,A -85,B 0,C 180,E1 27086.417,E2 27086.417} C_VEL
LIN {X 0,Y 559.95,Z 1170.699,A -85,B 0,C 180,E1 27083.644,E2 27083.644} C_VEL
LIN {X 0,Y 560.033,Z 1166.42,A -85,B 0,C 180,E1 27081.064,E2 27081.064} C_VEL
LIN {X 0,Y 560.202,Z 1161.195,A -85,B 0,C 180,E1 27078.678,E2 27078.678} C_VEL
LIN {X 0,Y 560.547,Z 1154.691,A -85,B 0,C 180,E1 27076.277,E2 27076.277} C_VEL
LIN {X 0,Y 561.238,Z 1144.902,A -85,B 0,C 180,E1 27073.332,E2 27073.332} C_VEL
LIN {X 0,Y 562.095,Z 1135.176,A -85,B 0,C 180,E1 27070.895,E2 27070.895} C_VEL
LIN {X 0,Y 563.131,Z 1125.476,A -85,B 0,C 180,E1 27068.764,E2 27068.764} C_VEL
LIN {X 0,Y 564.529,Z 1113.935,A -85,B 0,C 180,E1 27066.515,E2 27066.515} C_VEL
LIN {X 0,Y 566.674,Z 1098.16,A -85,B 0,C 180,E1 27063.825,E2 27063.825} C_VEL
LIN {X 0,Y 568.853,Z 1083.682,A -85,B 0,C 180,E1 27061.669,E2 27061.669} C_VEL
LIN {X 0,Y 571.144,Z 1069.157,A -85,B 0,C 180,E1 27059.723,E2 27059.723} C_VEL
LIN {X 0,Y 573.972,Z 1052.094,A -85,B 0,C 180,E1 27057.67,E2 27057.67} C_VEL
LIN {X 0,Y 577.535,Z 1031.13,A -85,B 0,C 180,E1 27055.46,E2 27055.46} C_VEL
LIN {X 0,Y 580.447,Z 1013.983,A -85,B 0,C 180,E1 27053.855,E2 27053.855} C_VEL
LIN {X 0,Y 583.37,Z 996.708,A -85,B 0,C 180,E1 27052.399,E2 27052.399} C_VEL
LIN {X 0,Y 586.535,Z 977.68,A -85,B 0,C 180,E1 27050.959,E2 27050.959} C_VEL
LIN {X 0,Y 590.423,Z 953.865,A -85,B 0,C 180,E1 27049.367,E2 27049.367} C_VEL
LIN {X 0,Y 593.693,Z 931.927,A -85,B 0,C 180,E1 27048.109,E2 27048.109} C_VEL
LIN {X 0,Y 596.323,Z 913.134,A -85,B 0,C 180,E1 27047.164,E2 27047.164} C_VEL
LIN {X 0,Y 598.768,Z 893.802,A -85,B 0,C 180,E1 27046.309,E2 27046.309} C_VEL
LIN {X 0,Y 601.153,Z 873.131,A -85,B 0,C 180,E1 27045.525,E2 27045.525} C_VEL
LIN {X 0,Y 603.311,Z 851.667,A -85,B 0,C 180,E1 27044.838,E2 27044.838} C_VEL
LIN {X 0,Y 605.603,Z 824.61,A -85,B 0,C 180,E1 27044.144,E2 27044.144} C_VEL
LIN {X 0,Y 607.139,Z 798.745,A -85,B 0,C 180,E1 27043.662,E2 27043.662} C_VEL
LIN {X 0,Y 610.753,Z 681.863,A -85,B 0,C 180,E1 27041.999,E2 27041.999} C_VEL
LIN {X 0,Y 617.49,Z 465.51,A -85,B 0,C 180,E1 27038.906,E2 27038.906} C_VEL
LIN {X 0,Y 619.305,Z 408.905,A -85,B 0,C 180,E1 27038.08,E2 27038.08} C_VEL
LIN {X 0,Y 605.449,Z 389.888,A -85,B 0,C 180,E1 27035.984,E2 27035.984} C_VEL
LIN {X 0,Y 596.918,Z 378.792,A -85,B 0,C 180,E1 27034.601,E2 27034.601} C_VEL
LIN {X 0,Y 589.425,Z 369.177,A -85,B 0,C 180,E1 27033.313,E2 27033.313} C_VEL
LIN {X 0,Y 584.516,Z 363.131,A -85,B 0,C 180,E1 27032.431,E2 27032.431} C_VEL
LIN {X 0,Y 580.658,Z 358.358,A -85,B 0,C 180,E1 27031.711,E2 27031.711} C_VEL
LIN {X 0,Y 577.097,Z 354.075,A -85,B 0,C 180,E1 27031.028,E2 27031.028} C_VEL
LIN {X 0,Y 575.743,Z 352.395,A -85,B 0,C 180,E1 27030.761,E2 27030.761} C_VEL
LIN {X 0,Y 572.483,Z 348.71,A -85,B 0,C 180,E1 27030.113,E2 27030.113} C_VEL
LIN {X 0,Y 571.315,Z 346.844,A -85,B 0,C 180,E1 27029.863,E2 27029.863} C_VEL
LIN {X 0,Y 568.192,Z 343.973,A -85,B 0,C 180,E1 27029.232,E2 27029.232} C_VEL
LIN {X 0,Y 566.371,Z 340.735,A -85,B 0,C 180,E1 27028.814,E2 27028.814} C_VEL
LIN {X 0,Y 563.284,Z 338.608,A -85,B 0,C 180,E1 27028.176,E2 27028.176} C_VEL
LIN {X 0,Y 561.67,Z 335.701,A -85,B 0,C 180,E1 27027.786,E2 27027.786} C_VEL
LIN {X 0,Y 561.379,Z 334.301,A -85,B 0,C 180,E1 27027.675,E2 27027.675} C_VEL
LIN {X 0,Y 561.347,Z 334.27,A -85,B 0,C 180,E1 27024.409,E2 27024.409} C_VEL
LIN {X 0,Y 561.393,Z 334.259,A -85,B 0,C 180,E1 27021.415,E2 27021.415} C_VEL
LIN {X 0,Y 561.357,Z 334.299,A -85,B 0,C 180,E1 27018.162,E2 27018.162} C_VEL
LIN {X 0,Y 561.432,Z 334.241,A -85,B 0,C 180,E1 27014.966,E2 27014.966} C_VEL
LIN {X 0,Y 561.365,Z 334.305,A -85,B 0,C 180,E1 27011.82,E2 27011.82} C_VEL
LIN {X 0,Y 561.408,Z 334.243,A -85,B 0,C 180,E1 27008.604,E2 27008.604} C_VEL
LIN {X 0,Y 561.372,Z 334.305,A -85,B 0,C 180,E1 27005.622,E2 27005.622} C_VEL
LIN {X 0,Y 561.4,Z 334.245,A -85,B 0,C 180,E1 27002.348,E2 27002.348} C_VEL
LIN {X 0,Y 561.388,Z 334.301,A -85,B 0,C 180,E1 26999.286,E2 26999.286} C_VEL
LIN {X 0,Y 561.381,Z 334.252,A -85,B 0,C 180,E1 26995.863,E2 26995.863} C_VEL
LIN {X 0,Y 561.433,Z 334.28,A -85,B 0,C 180,E1 26992.729,E2 26992.729} C_VEL
LIN {X 0,Y 561.381,Z 334.264,A -85,B 0,C 180,E1 26989.429,E2 26989.429} C_VEL
LIN {X 0,Y 561.44,Z 334.255,A -85,B 0,C 180,E1 26986.193,E2 26986.193} C_VEL
LIN {X 0,Y 561.399,Z 334.291,A -85,B 0,C 180,E1 26983.016,E2 26983.016} C_VEL
LIN {X 0,Y 561.41,Z 334.247,A -85,B 0,C 180,E1 26979.678,E2 26979.678} C_VEL
LIN {X 0,Y 561.43,Z 334.28,A -85,B 0,C 180,E1 26976.488,E2 26976.488} C_VEL
LIN {X 0,Y 561.456,Z 334.415,A -85,B 0,C 180,E1 26973.79,E2 26973.79} C_VEL
LIN {X 0,Y 562.763,Z 337.852,A -85,B 0,C 180,E1 26973.059,E2 26973.059} C_VEL
LIN {X 0,Y 564.21,Z 339.496,A -85,B 0,C 180,E1 26972.563,E2 26972.563} C_VEL
LIN {X 0,Y 565.943,Z 343.318,A -85,B 0,C 180,E1 26971.738,E2 26971.738} C_VEL
LIN {X 0,Y 567.159,Z 345.104,A -85,B 0,C 180,E1 26971.345,E2 26971.345} C_VEL
LIN {X 0,Y 570.479,Z 349.414,A -85,B 0,C 180,E1 26970.638,E2 26970.638} C_VEL
LIN {X 0,Y 580.211,Z 361.888,A -85,B 0,C 180,E1 26968.696,E2 26968.696} C_VEL
LIN {X 0,Y 589.503,Z 374.229,A -85,B 0,C 180,E1 26966.983,E2 26966.983} C_VEL
LIN {X 0,Y 599.562,Z 388.275,A -85,B 0,C 180,E1 26965.254,E2 26965.254} C_VEL
LIN {X 0,Y 611.143,Z 405.121,A -85,B 0,C 180,E1 26963.405,E2 26963.405} C_VEL
LIN {X 0,Y 619.541,Z 418.384,A -85,B 0,C 180,E1 26962.135,E2 26962.135} C_VEL
LIN {X 0,Y 612.866,Z 631.383,A -85,B 0,C 180,E1 26959.07,E2 26959.07} C_VEL
LIN {X 0,Y 607.028,Z 825.486,A -85,B 0,C 180,E1 26956.319,E2 26956.319} C_VEL
LIN {X 0,Y 605.603,Z 849.339,A -85,B 0,C 180,E1 26955.888,E2 26955.888} C_VEL
LIN {X 0,Y 603.251,Z 878.22,A -85,B 0,C 180,E1 26955.177,E2 26955.177} C_VEL
LIN {X 0,Y 601.057,Z 900.237,A -85,B 0,C 180,E1 26954.487,E2 26954.487} C_VEL
LIN {X 0,Y 598.677,Z 921.264,A -85,B 0,C 180,E1 26953.704,E2 26953.704} C_VEL
LIN {X 0,Y 596.254,Z 940.956,A -85,B 0,C 180,E1 26952.849,E2 26952.849} C_VEL
LIN {X 0,Y 593.502,Z 961.213,A -85,B 0,C 180,E1 26951.846,E2 26951.846} C_VEL
LIN {X 0,Y 589.905,Z 986.168,A -85,B 0,C 180,E1 26950.421,E2 26950.421} C_VEL
LIN {X 0,Y 586.375,Z 1008.483,A -85,B 0,C 180,E1 26948.934,E2 26948.934} C_VEL
LIN {X 0,Y 583.451,Z 1026.223,A -85,B 0,C 180,E1 26947.595,E2 26947.595} C_VEL
LIN {X 0,Y 580.646,Z 1042.828,A -85,B 0,C 180,E1 26946.202,E2 26946.202} C_VEL
LIN {X 0,Y 577.785,Z 1059.605,A -85,B 0,C 180,E1 26944.643,E2 26944.643} C_VEL
LIN {X 0,Y 574.6,Z 1078.508,A -85,B 0,C 180,E1 26942.687,E2 26942.687} C_VEL
LIN {X 0,Y 571.336,Z 1097.984,A -85,B 0,C 180,E1 26940.382,E2 26940.382} C_VEL
LIN {X 0,Y 569.021,Z 1112.608,A -85,B 0,C 180,E1 26938.437,E2 26938.437} C_VEL
LIN {X 0,Y 566.887,Z 1126.666,A -85,B 0,C 180,E1 26936.359,E2 26936.359} C_VEL
LIN {X 0,Y 564.72,Z 1142.546,A -85,B 0,C 180,E1 26933.698,E2 26933.698} C_VEL
LIN {X 0,Y 563.223,Z 1154.749,A -85,B 0,C 180,E1 26931.341,E2 26931.341} C_VEL
LIN {X 0,Y 562.124,Z 1164.984,A -85,B 0,C 180,E1 26929.104,E2 26929.104} C_VEL
LIN {X 0,Y 561.248,Z 1174.731,A -85,B 0,C 180,E1 26926.668,E2 26926.668} C_VEL
LIN {X 0,Y 560.562,Z 1184.561,A -85,B 0,C 180,E1 26923.723,E2 26923.723} C_VEL
LIN {X 0,Y 560.206,Z 1191.085,A -85,B 0,C 180,E1 26921.322,E2 26921.322} C_VEL
LIN {X 0,Y 560.034,Z 1196.33,A -85,B 0,C 180,E1 26918.936,E2 26918.936} C_VEL
LIN {X 0,Y 559.945,Z 1200.782,A -85,B 0,C 180,E1 26916.253,E2 26916.253} C_VEL
LIN {X 0,Y 559.914,Z 1203.641,A -85,B 0,C 180,E1 26913.481,E2 26913.481} C_VEL
LIN {X 0,Y 559.916,Z 1204.736,A -85,B 0,C 180,E1 26911.228,E2 26911.228} C_VEL
LIN {X 0,Y 559.906,Z 1204.804,A -85,B 0,C 180,E1 26909.079,E2 26909.079} C_VEL
LIN {X 0,Y 559.917,Z 1203.845,A -85,B 0,C 180,E1 26906.827,E2 26906.827} C_VEL
LIN {X 0,Y 559.933,Z 1201.534,A -85,B 0,C 180,E1 26904.364,E2 26904.364} C_VEL
LIN {X 0,Y 560.017,Z 1197.151,A -85,B 0,C 180,E1 26901.478,E2 26901.478} C_VEL
LIN {X 0,Y 560.181,Z 1191.594,A -85,B 0,C 180,E1 26898.886,E2 26898.886} C_VEL
LIN {X 0,Y 560.532,Z 1185.077,A -85,B 0,C 180,E1 26896.456,E2 26896.456} C_VEL
LIN {X 0,Y 561.163,Z 1175.941,A -85,B 0,C 180,E1 26893.649,E2 26893.649} C_VEL
LIN {X 0,Y 562.082,Z 1165.446,A -85,B 0,C 180,E1 26891.002,E2 26891.002} C_VEL
LIN {X 0,Y 563.161,Z 1155.269,A -85,B 0,C 180,E1 26888.765,E2 26888.765} C_VEL
LIN {X 0,Y 564.639,Z 1143.132,A -85,B 0,C 180,E1 26886.409,E2 26886.409} C_VEL
LIN {X 0,Y 566.813,Z 1127.181,A -85,B 0,C 180,E1 26883.72,E2 26883.72} C_VEL
LIN {X 0,Y 569.021,Z 1112.608,A -85,B 0,C 180,E1 26881.563,E2 26881.563} C_VEL
LIN {X 0,Y 571.336,Z 1097.984,A -85,B 0,C 180,E1 26879.618,E2 26879.618} C_VEL
LIN {X 0,Y 574.6,Z 1078.508,A -85,B 0,C 180,E1 26877.313,E2 26877.313} C_VEL
LIN {X 0,Y 577.784,Z 1059.604,A -85,B 0,C 180,E1 26875.356,E2 26875.356} C_VEL
LIN {X 0,Y 580.645,Z 1042.823,A -85,B 0,C 180,E1 26873.798,E2 26873.798} C_VEL
LIN {X 0,Y 583.449,Z 1026.214,A -85,B 0,C 180,E1 26872.405,E2 26872.405} C_VEL
LIN {X 0,Y 586.457,Z 1007.969,A -85,B 0,C 180,E1 26871.029,E2 26871.029} C_VEL
LIN {X 0,Y 590.155,Z 984.56,A -85,B 0,C 180,E1 26869.478,E2 26869.478} C_VEL
LIN {X 0,Y 593.588,Z 960.572,A -85,B 0,C 180,E1 26868.12,E2 26868.12} C_VEL
LIN {X 0,Y 596.254,Z 940.96,A -85,B 0,C 180,E1 26867.151,E2 26867.151} C_VEL
LIN {X 0,Y 598.678,Z 921.265,A -85,B 0,C 180,E1 26866.296,E2 26866.296} C_VEL
LIN {X 0,Y 601.058,Z 900.239,A -85,B 0,C 180,E1 26865.513,E2 26865.513} C_VEL
LIN {X 0,Y 603.414,Z 876.647,A -85,B 0,C 180,E1 26864.778,E2 26864.778} C_VEL
LIN {X 0,Y 605.671,Z 848.205,A -85,B 0,C 180,E1 26864.089,E2 26864.089} C_VEL
LIN {X 0,Y 607.049,Z 825.027,A -85,B 0,C 180,E1 26863.674,E2 26863.674} C_VEL
LIN {X 0,Y 613.163,Z 621.418,A -85,B 0,C 180,E1 26860.788,E2 26860.788} C_VEL
LIN {X 0,Y 619.541,Z 418.075,A -85,B 0,C 180,E1 26857.862,E2 26857.862} C_VEL
LIN {X 0,Y 606.394,Z 398.142,A -85,B 0,C 180,E1 26855.858,E2 26855.858} C_VEL
LIN {X 0,Y 593.595,Z 379.832,A -85,B 0,C 180,E1 26853.742,E2 26853.742} C_VEL
LIN {X 0,Y 582.83,Z 365.324,A -85,B 0,C 180,E1 26851.811,E2 26851.811} C_VEL
LIN {X 0,Y 577.188,Z 358.057,A -85,B 0,C 180,E1 26850.733,E2 26850.733} C_VEL
LIN {X 0,Y 570.419,Z 349.356,A -85,B 0,C 180,E1 26849.365,E2 26849.365} C_VEL
LIN {X 0,Y 567.098,Z 345.002,A -85,B 0,C 180,E1 26848.658,E2 26848.658} C_VEL
LIN {X 0,Y 564.498,Z 340.554,A -85,B 0,C 180,E1 26847.651,E2 26847.651} C_VEL
LIN {X 0,Y 563.762,Z 339.027,A -85,B 0,C 180,E1 26847.309,E2 26847.309} C_VEL
LIN {X 0,Y 561.84,Z 336.029,A -85,B 0,C 180,E1 26846.532,E2 26846.532} C_VEL
LIN {X 0,Y 561.436,Z 334.255,A -85,B 0,C 180,E1 26846.16,E2 26846.16} C_VEL
LIN {X 0,Y 561.401,Z 334.303,A -85,B 0,C 180,E1 26842.847,E2 26842.847} C_VEL
LIN {X 0,Y 561.435,Z 334.248,A -85,B 0,C 180,E1 26839.562,E2 26839.562} C_VEL
LIN {X 0,Y 561.402,Z 334.271,A -85,B 0,C 180,E1 26836.344,E2 26836.344} C_VEL
LIN {X 0,Y 561.4,Z 334.281,A -85,B 0,C 180,E1 26832.969,E2 26832.969} C_VEL
LIN {X 0,Y 561.423,Z 334.248,A -85,B 0,C 180,E1 26829.845,E2 26829.845} C_VEL
LIN {X 0,Y 561.388,Z 334.302,A -85,B 0,C 180,E1 26826.545,E2 26826.545} C_VEL
LIN {X 0,Y 561.434,Z 334.24,A -85,B 0,C 180,E1 26823.369,E2 26823.369} C_VEL
LIN {X 0,Y 561.381,Z 334.302,A -85,B 0,C 180,E1 26820.204,E2 26820.204} C_VEL
LIN {X 0,Y 561.411,Z 334.242,A -85,B 0,C 180,E1 26816.937,E2 26816.937} C_VEL
LIN {X 0,Y 561.382,Z 334.303,A -85,B 0,C 180,E1 26813.865,E2 26813.865} C_VEL
LIN {X 0,Y 561.377,Z 334.25,A -85,B 0,C 180,E1 26810.465,E2 26810.465} C_VEL
LIN {X 0,Y 561.406,Z 334.292,A -85,B 0,C 180,E1 26807.346,E2 26807.346} C_VEL
LIN {X 0,Y 561.362,Z 334.26,A -85,B 0,C 180,E1 26804.114,E2 26804.114} C_VEL
LIN {X 0,Y 561.422,Z 334.267,A -85,B 0,C 180,E1 26800.978,E2 26800.978} C_VEL
LIN {X 0,Y 561.354,Z 334.283,A -85,B 0,C 180,E1 26797.814,E2 26797.814} C_VEL
LIN {X 0,Y 561.419,Z 334.249,A -85,B 0,C 180,E1 26794.695,E2 26794.695} C_VEL
LIN {X 0,Y 561.398,Z 334.469,A -85,B 0,C 180,E1 26792.191,E2 26792.191} C_VEL
LIN {X 0,Y 562.392,Z 337.357,A -85,B 0,C 180,E1 26791.92,E2 26791.92} C_VEL
LIN {X 0,Y 564.82,Z 339.935,A -85,B 0,C 180,E1 26791.389,E2 26791.389} C_VEL
LIN {X 0,Y 566.657,Z 341.183,A -85,B 0,C 180,E1 26791.014,E2 26791.014} C_VEL
LIN {X 0,Y 568.871,Z 344.82,A -85,B 0,C 180,E1 26790.518,E2 26790.518} C_VEL
LIN {X 0,Y 571.789,Z 347.491,A -85,B 0,C 180,E1 26789.933,E2 26789.933} C_VEL
LIN {X 0,Y 574.75,Z 351.508,A -85,B 0,C 180,E1 26789.325,E2 26789.325} C_VEL
LIN {X 0,Y 576.711,Z 353.434,A -85,B 0,C 180,E1 26788.949,E2 26788.949} C_VEL
LIN {X 0,Y 580.123,Z 357.866,A -85,B 0,C 180,E1 26788.285,E2 26788.285} C_VEL
LIN {X 0,Y 582.118,Z 360.109,A -85,B 0,C 180,E1 26787.914,E2 26787.914} C_VEL
LIN {X 0,Y 586.961,Z 366.195,A -85,B 0,C 180,E1 26787.025,E2 26787.025} C_VEL
LIN {X 0,Y 591.934,Z 372.366,A -85,B 0,C 180,E1 26786.15,E2 26786.15} C_VEL
LIN {X 0,Y 602.712,Z 386.211,A -85,B 0,C 180,E1 26784.358,E2 26784.358} C_VEL
LIN {X 0,Y 614.584,Z 402.408,A -85,B 0,C 180,E1 26782.52,E2 26782.52} C_VEL
LIN {X 0,Y 619.327,Z 409.213,A -85,B 0,C 180,E1 26781.821,E2 26781.821} C_VEL
LIN {X 0,Y 612.33,Z 629.574,A -85,B 0,C 180,E1 26778.652,E2 26778.652} C_VEL
LIN {X 0,Y 610.104,Z 703.745,A -85,B 0,C 180,E1 26777.601,E2 26777.601} C_VEL
LIN {X 0,Y 609.201,Z 711.447,A -85,B 0,C 180,E1 26777.563,E2 26777.563} C_VEL
LIN {X 0,Y 604.396,Z 732.084,A -85,B 0,C 180,E1 26777.708,E2 26777.708} C_VEL
LIN {X 0,Y 603.673,Z 738.694,A -85,B 0,C 180,E1 26777.669,E2 26777.669} C_VEL
LIN {X 0,Y 601.543,Z 800.958,A -85,B 0,C 180,E1 26776.768,E2 26776.768} C_VEL
LIN {X 0,Y 599.613,Z 829.895,A -85,B 0,C 180,E1 26776.199,E2 26776.199} C_VEL
LIN {X 0,Y 597.494,Z 853.531,A -85,B 0,C 180,E1 26775.572,E2 26775.572} C_VEL
LIN {X 0,Y 595.311,Z 874.312,A -85,B 0,C 180,E1 26774.897,E2 26774.897} C_VEL
LIN {X 0,Y 592.849,Z 894.756,A -85,B 0,C 180,E1 26774.113,E2 26774.113} C_VEL
LIN {X 0,Y 589.983,Z 916.362,A -85,B 0,C 180,E1 26773.143,E2 26773.143} C_VEL
LIN {X 0,Y 586.109,Z 942.193,A -85,B 0,C 180,E1 26771.778,E2 26771.778} C_VEL
LIN {X 0,Y 582.716,Z 962.894,A -85,B 0,C 180,E1 26770.5,E2 26770.5} C_VEL
LIN {X 0,Y 579.587,Z 981.111,A -85,B 0,C 180,E1 26769.23,E2 26769.23} C_VEL
LIN {X 0,Y 576.502,Z 998.487,A -85,B 0,C 180,E1 26767.876,E2 26767.876} C_VEL
LIN {X 0,Y 572.507,Z 1020.871,A -85,B 0,C 180,E1 26765.931,E2 26765.931} C_VEL
LIN {X 0,Y 568.911,Z 1040.664,A -85,B 0,C 180,E1 26763.946,E2 26763.946} C_VEL
LIN {X 0,Y 566.18,Z 1056.037,A -85,B 0,C 180,E1 26762.228,E2 26762.228} C_VEL
LIN {X 0,Y 563.582,Z 1071.04,A -85,B 0,C 180,E1 26760.373,E2 26760.373} C_VEL
LIN {X 0,Y 560.783,Z 1087.951,A -85,B 0,C 180,E1 26758.042,E2 26758.042} C_VEL
LIN {X 0,Y 558.286,Z 1104.025,A -85,B 0,C 180,E1 26755.489,E2 26755.489} C_VEL
LIN {X 0,Y 556.543,Z 1116.34,A -85,B 0,C 180,E1 26753.281,E2 26753.281} C_VEL
LIN {X 0,Y 555.062,Z 1128.146,A -85,B 0,C 180,E1 26750.896,E2 26750.896} C_VEL
LIN {X 0,Y 553.743,Z 1140.512,A -85,B 0,C 180,E1 26747.985,E2 26747.985} C_VEL
LIN {X 0,Y 552.988,Z 1149.006,A -85,B 0,C 180,E1 26745.629,E2 26745.629} C_VEL
LIN {X 0,Y 552.506,Z 1156.247,A -85,B 0,C 180,E1 26743.287,E2 26743.287} C_VEL
LIN {X 0,Y 552.164,Z 1163.003,A -85,B 0,C 180,E1 26740.644,E2 26740.644} C_VEL
LIN {X 0,Y 551.987,Z 1168.59,A -85,B 0,C 180,E1 26737.751,E2 26737.751} C_VEL
LIN {X 0,Y 551.928,Z 1171.937,A -85,B 0,C 180,E1 26735.301,E2 26735.301} C_VEL
LIN {X 0,Y 551.912,Z 1174.017,A -85,B 0,C 180,E1 26732.908,E2 26732.908} C_VEL
LIN {X 0,Y 551.894,Z 1174.885,A -85,B 0,C 180,E1 26730.519,E2 26730.519} C_VEL
LIN {X 0,Y 551.909,Z 1174.407,A -85,B 0,C 180,E1 26727.612,E2 26727.612} C_VEL
LIN {X 0,Y 551.922,Z 1172.377,A -85,B 0,C 180,E1 26725.011,E2 26725.011} C_VEL
LIN {X 0,Y 551.974,Z 1169.281,A -85,B 0,C 180,E1 26722.611,E2 26722.611} C_VEL
LIN {X 0,Y 552.092,Z 1164.862,A -85,B 0,C 180,E1 26720.144,E2 26720.144} C_VEL
LIN {X 0,Y 552.405,Z 1158.012,A -85,B 0,C 180,E1 26717.243,E2 26717.243} C_VEL
LIN {X 0,Y 552.898,Z 1150.363,A -85,B 0,C 180,E1 26714.691,E2 26714.691} C_VEL
LIN {X 0,Y 553.548,Z 1142.467,A -85,B 0,C 180,E1 26712.444,E2 26712.444} C_VEL
LIN {X 0,Y 554.477,Z 1133.335,A -85,B 0,C 180,E1 26710.183,E2 26710.183} C_VEL
LIN {X 0,Y 555.98,Z 1120.802,A -85,B 0,C 180,E1 26707.477,E2 26707.477} C_VEL
LIN {X 0,Y 557.892,Z 1106.613,A -85,B 0,C 180,E1 26704.865,E2 26704.865} C_VEL
LIN {X 0,Y 559.818,Z 1093.949,A -85,B 0,C 180,E1 26702.792,E2 26702.792} C_VEL
LIN {X 0,Y 562.216,Z 1079.05,A -85,B 0,C 180,E1 26700.604,E2 26700.604} C_VEL
LIN {X 0,Y 565.595,Z 1059.495,A -85,B 0,C 180,E1 26698.091,E2 26698.091} C_VEL
LIN {X 0,Y 568.466,Z 1043.168,A -85,B 0,C 180,E1 26696.234,E2 26696.234} C_VEL
LIN {X 0,Y 571.43,Z 1026.68,A -85,B 0,C 180,E1 26694.547,E2 26694.547} C_VEL
LIN {X 0,Y 574.934,Z 1007.181,A -85,B 0,C 180,E1 26692.757,E2 26692.757} C_VEL
LIN {X 0,Y 578.995,Z 984.483,A -85,B 0,C 180,E1 26690.927,E2 26690.927} C_VEL
LIN {X 0,Y 582.243,Z 965.627,A -85,B 0,C 180,E1 26689.589,E2 26689.589} C_VEL
LIN {X 0,Y 585.275,Z 947.164,A -85,B 0,C 180,E1 26688.424,E2 26688.424} C_VEL
LIN {X 0,Y 588.365,Z 927.152,A -85,B 0,C 180,E1 26687.308,E2 26687.308} C_VEL
LIN {X 0,Y 591.959,Z 902.134,A -85,B 0,C 180,E1 26686.103,E2 26686.103} C_VEL
LIN {X 0,Y 595.007,Z 876.997,A -85,B 0,C 180,E1 26685.108,E2 26685.108} C_VEL
LIN {X 0,Y 597.281,Z 855.71,A -85,B 0,C 180,E1 26684.404,E2 26684.404} C_VEL
LIN {X 0,Y 599.218,Z 834.592,A -85,B 0,C 180,E1 26683.828,E2 26683.828} C_VEL
LIN {X 0,Y 600.857,Z 812.439,A -85,B 0,C 180,E1 26683.344,E2 26683.344} C_VEL
LIN {X 0,Y 602.384,Z 781.046,A -85,B 0,C 180,E1 26682.84,E2 26682.84} C_VEL
LIN {X 0,Y 609.444,Z 556.877,A -85,B 0,C 180,E1 26679.643,E2 26679.643} C_VEL
LIN {X 0,Y 614.181,Z 413.034,A -85,B 0,C 180,E1 26677.539,E2 26677.539} C_VEL
LIN {X 0,Y 601.774,Z 395.958,A -85,B 0,C 180,E1 26675.618,E2 26675.618} C_VEL
LIN {X 0,Y 593.597,Z 385.209,A -85,B 0,C 180,E1 26674.266,E2 26674.266} C_VEL
LIN {X 0,Y 586.297,Z 375.798,A -85,B 0,C 180,E1 26672.988,E2 26672.988} C_VEL
LIN {X 0,Y 580.969,Z 369.209,A -85,B 0,C 180,E1 26672.012,E2 26672.012} C_VEL
LIN {X 0,Y 577.616,Z 365.066,A -85,B 0,C 180,E1 26671.374,E2 26671.374} C_VEL
LIN {X 0,Y 573.895,Z 360.288,A -85,B 0,C 180,E1 26670.639,E2 26670.639} C_VEL
LIN {X 0,Y 569.764,Z 355.608,A -85,B 0,C 180,E1 26669.807,E2 26669.807} C_VEL
LIN {X 0,Y 568.362,Z 353.77,A -85,B 0,C 180,E1 26669.511,E2 26669.511} C_VEL
LIN {X 0,Y 565.109,Z 350.247,A -85,B 0,C 180,E1 26668.826,E2 26668.826} C_VEL
LIN {X 0,Y 563.682,Z 348.013,A -85,B 0,C 180,E1 26668.501,E2 26668.501} C_VEL
LIN {X 0,Y 560.466,Z 345.248,A -85,B 0,C 180,E1 26667.809,E2 26667.809} C_VEL
LIN {X 0,Y 558.331,Z 341.659,A -85,B 0,C 180,E1 26667.288,E2 26667.288} C_VEL
LIN {X 0,Y 555.206,Z 339.392,A -85,B 0,C 180,E1 26666.586,E2 26666.586} C_VEL
LIN {X 0,Y 553.693,Z 336.605,A -85,B 0,C 180,E1 26666.187,E2 26666.187} C_VEL
LIN {X 0,Y 553.406,Z 335.247,A -85,B 0,C 180,E1 26666.072,E2 26666.072} C_VEL
LIN {X 0,Y 553.438,Z 335.292,A -85,B 0,C 180,E1 26662.745,E2 26662.745} C_VEL
LIN {X 0,Y 553.423,Z 335.241,A -85,B 0,C 180,E1 26659.733,E2 26659.733} C_VEL
LIN {X 0,Y 553.425,Z 335.264,A -85,B 0,C 180,E1 26656.371,E2 26656.371} C_VEL
LIN {X 0,Y 553.449,Z 335.253,A -85,B 0,C 180,E1 26653.371,E2 26653.371} C_VEL
LIN {X 0,Y 553.423,Z 335.25,A -85,B 0,C 180,E1 26650.056,E2 26650.056} C_VEL
LIN {X 0,Y 553.506,Z 335.265,A -85,B 0,C 180,E1 26646.848,E2 26646.848} C_VEL
LIN {X 0,Y 553.427,Z 335.241,A -85,B 0,C 180,E1 26643.626,E2 26643.626} C_VEL
LIN {X 0,Y 553.47,Z 335.281,A -85,B 0,C 180,E1 26640.311,E2 26640.311} C_VEL
LIN {X 0,Y 553.447,Z 335.235,A -85,B 0,C 180,E1 26637.204,E2 26637.204} C_VEL
LIN {X 0,Y 553.448,Z 335.289,A -85,B 0,C 180,E1 26633.777,E2 26633.777} C_VEL
LIN {X 0,Y 553.49,Z 335.227,A -85,B 0,C 180,E1 26630.643,E2 26630.643} C_VEL
LIN {X 0,Y 553.449,Z 335.285,A -85,B 0,C 180,E1 26627.373,E2 26627.373} C_VEL
LIN {X 0,Y 553.492,Z 335.24,A -85,B 0,C 180,E1 26624.062,E2 26624.062} C_VEL
LIN {X 0,Y 553.463,Z 335.249,A -85,B 0,C 180,E1 26620.878,E2 26620.878} C_VEL
LIN {X 0,Y 553.467,Z 335.286,A -85,B 0,C 180,E1 26617.48,E2 26617.48} C_VEL
LIN {X 0,Y 553.479,Z 335.395,A -85,B 0,C 180,E1 26615.283,E2 26615.283} C_VEL
LIN {X 0,Y 554.854,Z 338.815,A -85,B 0,C 180,E1 26614.488,E2 26614.488} C_VEL
LIN {X 0,Y 556.405,Z 340.861,A -85,B 0,C 180,E1 26613.878,E2 26613.878} C_VEL
LIN {X 0,Y 558.19,Z 344.478,A -85,B 0,C 180,E1 26613.079,E2 26613.079} C_VEL
LIN {X 0,Y 560.128,Z 346.718,A -85,B 0,C 180,E1 26612.634,E2 26612.634} C_VEL
LIN {X 0,Y 563.65,Z 350.986,A -85,B 0,C 180,E1 26611.844,E2 26611.844} C_VEL
LIN {X 0,Y 568.215,Z 356.776,A -85,B 0,C 180,E1 26610.856,E2 26610.856} C_VEL
LIN {X 0,Y 577.628,Z 369.122,A -85,B 0,C 180,E1 26608.946,E2 26608.946} C_VEL
LIN {X 0,Y 586.608,Z 381.123,A -85,B 0,C 180,E1 26607.264,E2 26607.264} C_VEL
LIN {X 0,Y 598.833,Z 398.354,A -85,B 0,C 180,E1 26605.147,E2 26605.147} C_VEL
LIN {X 0,Y 611.701,Z 417.784,A -85,B 0,C 180,E1 26603.093,E2 26603.093} C_VEL
LIN {X 0,Y 614.477,Z 422.434,A -85,B 0,C 180,E1 26602.665,E2 26602.665} C_VEL
LIN {X 0,Y 607.444,Z 636.583,A -85,B 0,C 180,E1 26599.566,E2 26599.566} C_VEL
LIN {X 0,Y 601.492,Z 825.292,A -85,B 0,C 180,E1 26596.873,E2 26596.873} C_VEL
